// TwinCAT 3 PLC project PLC_v01
// ProgramVersion: 3.1.4022.1
// libraries:
//   Tc2_MC2, * (Beckhoff Automation GmbH)
//   Tc2_MC2_Drive, * (Beckhoff Automation GmbH)
//   Tc2_NCI, * (Beckhoff Automation GmbH)
//   Tc2_NcKinematicTransformation, * (Beckhoff Automation GmbH)
//   Tc2_Standard, * (Beckhoff Automation GmbH)
//   Tc2_System, * (Beckhoff Automation GmbH)
//   Tc2_Utilities, * (Beckhoff Automation GmbH)
//   Tc3_Module, * (Beckhoff Automation GmbH)
//   Tc3_PLCopen_OpcUa, * (Beckhoff Automation GmbH)
//   VisuDialogs, * (System)
// project tree:
//   DUTs/ E_NciChannelState.TcDUT (not stored), ST_AxisInterface.TcDUT (not stored), ST_AxisInterfaceIn.TcDUT (not stored), ST_AxisInterfaceOut.TcDUT (not stored), ST_FileDialogParams.TcDUT (not stored), ST_OpcUAVariablesR.TcDUT (not stored), ST_OpcUAVariablesW.TcDUT
//   GVLs/ GVL_Axis.TcGVL, GVL_FileOpen.TcGVL, GVL_Kin.TcGVL (not stored), GVL_Nci.TcGVL (not stored), GVL_Process.TcGVL
//   / PlcTask.TcTTO (not stored), Visualization Manager.TcVMO (not stored)
//   POUs/ FB_AxisControl.TcPOU, MAIN.TcPOU, PRG_MFuncControl.TcPOU, PRG_NcControl.TcPOU (not stored), PRG_Process.TcPOU
//   POUs/KIN/ PRG_Kinematic.TcPOU (not stored)
//   POUs/NCI/ FB_NciChannel.TcPOU, FB_NciFastMFunctions.TcPOU (not stored), FB_NciMFunctions.TcPOU, FB_NciReadLine.TcPOU, FB_NciWriteToolParams.TcPOU
//   POUs/OPC-UA/ FB_OpcUAWrite.TcPOU, PRG_OpcUA.TcPOU
//   POUs/UTIL/ FB_Flash.TcPOU, FB_ScreenOnOff_Win7.TcPOU (not stored)
//   VISUs/AxisList/ VisuAxisM1.TcVIS (not stored), VisuAxisM2.TcVIS (not stored), VisuAxisM3.TcVIS (not stored), VisuAxisX.TcVIS, VisuAxisX_1.TcVIS (not stored), VisuAxisY.TcVIS (not stored), VisuAxisY_1.TcVIS (not stored), VisuAxisZ.TcVIS, VisuAxisZ_1.TcVIS
//   VISUs/Frame/ Visualization_FileList.TcVIS (not stored), VisuAxisControl.TcVIS (not stored), VisuAxisControl_1.TcVIS (not stored), VisuAxisInfo.TcVIS
//   VISUs/ GlobalTextList.TcGTLO, ImagePool.TcIPO (not stored), Visualization.TcVIS, Visualization_AxesInfo.TcVIS (not stored), Visualization_AxesInfo_Manual.TcVIS (not stored)
// real-time tasks:
//   TASK PlcTask: cycle T#10ms, priority 20, ADS port 350
// motion (NC):
//   TASK NC-Task 1 SAF: cycle T#2ms, priority 4, ADS port 501
//   TASK NC-Task 1 SVB: cycle T#10ms, priority 8, ADS port 511
//   AXIS M1 (id 1)
//     Dynamic: Acceleration=120.483870963794, Deceleration=120.483870963794, Jerk=361.451612891381, DelayTime=0.008
//     Velo: RefSearch=0.803225806425292, RefSync=0.803225806425292, SlowManual=10, FastManual=25, Fast=80.3225806425291, Maximum=80.3225806425291
//     OtherSettings: AllowMotionCmdToSlave=true
//     encoder EncType=1
//       EncPara: ScaleFactorNumerator=11.6129032254259, ScaleFactorDenominator=1048576, Offset=-0.7867, Inverse=true
//     drive DrvType=5
//       DrvPara: Inverse=true
//         Analog: VeloReferenz=88.3548387067821, TorqueScale=10, ScaleFactorActTorque=0.1
//         TimeComp: TaskDelayCycles=1
//     controller CtrType=1
//       CtrPara: PriorControlFactor=1
//         PID: PosKp=10
//         Observer: BandWidth=20
//   AXIS M2 (id 2)
//     Dynamic: Acceleration=120.483870963794, Deceleration=120.483870963794, Jerk=361.451612891381, DelayTime=0.008
//     Velo: RefSearch=0.803225806425292, RefSync=0.803225806425292, SlowManual=10, FastManual=25, Fast=80.3225806425291, Maximum=80.3225806425291
//     OtherSettings: AllowMotionCmdToSlave=true
//     encoder EncType=1
//       EncPara: ScaleFactorNumerator=11.6129032254259, ScaleFactorDenominator=1048576, Offset=-4.6881, Inverse=true
//     drive DrvType=5
//       DrvPara: Inverse=true
//         Analog: VeloReferenz=88.3548387067821, TorqueScale=10, ScaleFactorActTorque=0.1
//         TimeComp: TaskDelayCycles=1
//     controller CtrType=1
//       CtrPara: PriorControlFactor=1
//         PID: PosKp=10
//         Observer: BandWidth=20
//   AXIS M3 (id 3)
//     Dynamic: Acceleration=120.483870963794, Deceleration=120.483870963794, Jerk=361.451612891381, DelayTime=0.008
//     Velo: RefSearch=0.803225806425292, RefSync=0.803225806425292, SlowManual=10, FastManual=25, Fast=80.3225806425291, Maximum=80.3225806425291
//     OtherSettings: AllowMotionCmdToSlave=true
//     encoder EncType=1
//       EncPara: ScaleFactorNumerator=11.6129032254259, ScaleFactorDenominator=1048576, Offset=4810.3626, Inverse=true
//     drive DrvType=5
//       DrvPara: Inverse=true
//         Analog: VeloReferenz=88.3548387067821, TorqueScale=10, ScaleFactorActTorque=0.1
//         TimeComp: TaskDelayCycles=1
//     controller CtrType=1
//       CtrPara: PriorControlFactor=1
//         PID: PosKp=10
//         Observer: BandWidth=20
//   AXIS X (id 4)
//     OtherSettings: AllowMotionCmdToSlave=true
//     encoder EncType=1
//     drive DrvType=5
//       Analog: ScaleFactorActTorque=0.1
//       TimeComp: TaskDelayCycles=1
//     controller CtrType=1
//       CtrPara: PriorControlFactor=1
//         Observer: BandWidth=20
//   AXIS Y (id 5)
//     OtherSettings: AllowMotionCmdToSlave=true
//     encoder EncType=1
//     drive DrvType=5
//       Analog: ScaleFactorActTorque=0.1
//       TimeComp: TaskDelayCycles=1
//     controller CtrType=1
//       CtrPara: PriorControlFactor=1
//         Observer: BandWidth=20
//   AXIS Z (id 6)
//     OtherSettings: AllowMotionCmdToSlave=true
//     encoder EncType=1
//     drive DrvType=5
//       Analog: ScaleFactorActTorque=0.1
//       TimeComp: TaskDelayCycles=1
//     controller CtrType=1
//       CtrPara: PriorControlFactor=1
//         Observer: BandWidth=20
// I/O:
//   DEVICE Device 1 (EtherCAT) (disabled), AmsNetId 10.70.16.23.2.1
//     Term 1 (EK1200) [EK1200-5000 EtherCAT Power supply (2A E-Bus)]
//       Term 2 (EL1008) [EL1008 8Ch. Dig. Input 24V, 3ms]
//       Term 3 (EL2008) [EL2008 8Ch. Dig. Output 24V, 0.5A]
//       Term 4 (EL9576) [EL9576 Brake chopper terminal]
//       Term 5 (EL7211-0010) [EL7211-0010 1Ch. MDP742 Servo motor output stage with OCT (50V, 4.5A RMS)]
//       Term 6 (EL7211-0010) [EL7211-0010 1Ch. MDP742 Servo motor output stage with OCT (50V, 4.5A RMS)]
//       Term 7 (EL7211-0010) [EL7211-0010 1Ch. MDP742 Servo motor output stage with OCT (50V, 4.5A RMS)]
//       Term 8 (EL9011) [EL9011 End Terminal]
// variable links:
//   PLC_v01/PLC_v01 Instance <-> NC-Task 1 SAF/Axes/M1
//     PlcTask Inputs/GVL_Axis.AxisM1_B.NcToPlc <-> Outputs/ToPlc
//     PlcTask Outputs/GVL_Axis.AxisM1_B.PlcToNc <-> Inputs/FromPlc
//   PLC_v01/PLC_v01 Instance <-> NC-Task 1 SAF/Axes/M2
//     PlcTask Inputs/GVL_Axis.AxisM2_C.NcToPlc <-> Outputs/ToPlc
//     PlcTask Outputs/GVL_Axis.AxisM2_C.PlcToNc <-> Inputs/FromPlc
//   PLC_v01/PLC_v01 Instance <-> NC-Task 1 SAF/Axes/M3
//     PlcTask Inputs/GVL_Axis.AxisM3_A.NcToPlc <-> Outputs/ToPlc
//     PlcTask Outputs/GVL_Axis.AxisM3_A.PlcToNc <-> Inputs/FromPlc
//   PLC_v01/PLC_v01 Instance <-> NC-Task 1 SAF/Axes/X
//     PlcTask Inputs/GVL_Axis.AxisX.NcToPlc <-> Outputs/ToPlc
//     PlcTask Outputs/GVL_Axis.AxisX.PlcToNc <-> Inputs/FromPlc
//   PLC_v01/PLC_v01 Instance <-> NC-Task 1 SAF/Axes/Y
//     PlcTask Inputs/GVL_Axis.AxisY.NcToPlc <-> Outputs/ToPlc
//     PlcTask Outputs/GVL_Axis.AxisY.PlcToNc <-> Inputs/FromPlc
//   PLC_v01/PLC_v01 Instance <-> NC-Task 1 SAF/Axes/Z
//     PlcTask Inputs/GVL_Axis.AxisZ.NcToPlc <-> Outputs/ToPlc
//     PlcTask Outputs/GVL_Axis.AxisZ.PlcToNc <-> Inputs/FromPlc
//   PLC_v01/PLC_v01 Instance <-> NC-Task 1 SAF/KIN
//     PlcTask Inputs/GVL_Kin.stKinToPLC <-> Outputs/ToPlc
//     PlcTask Outputs/GVL_Kin.stKinFromPLC <-> Inputs/FromPlc
//   PLC_v01/PLC_v01 Instance <-> NC-Task 1 SAF/NCI
//     PlcTask Inputs/GVL_Nci.stNciToPLC <-> Outputs/ToPlc
//     PlcTask Outputs/GVL_Nci.stPlcToNci <-> Inputs/FromPlc

// ---- DUTs/ST_OpcUAVariablesW.TcDUT
TYPE ST_OpcUAVariablesW :
STRUCT
	fActPosX		: LREAL;
	fActPosY		: LREAL;
	fActPosZ		: LREAL;
	fActPosM1		: LREAL;
	fActPosM2		: LREAL;
	fActPosM3		: LREAL;
	
	fActVeloX		: LREAL;
	fActVeloY		: LREAL;
	fActVeloZ		: LREAL;
	fActVeloM1		: LREAL;
	fActVeloM2		: LREAL;
	fActVeloM3		: LREAL;
	
	fLagDistanceX	: LREAL;
	fLagDistanceY	: LREAL;
	fLagDistanceZ	: LREAL;
	fLagDistanceM1	: LREAL;
	fLagDistanceM2	: LREAL;
	fLagDistanceM3	: LREAL;
	
	sNciActLine		: STRING;
	sNciLines		: STRING;
	sFileNameVisu	: STRING;
	
	bEnabledX		: BOOL;
	bEnabledY		: BOOL;
	bEnabledZ		: BOOL;
	bEnabledM1		: BOOL;
	bEnabledM2		: BOOL;
	bEnabledM3		: BOOL;
		
	bNciRunning		: BOOL;
	bNciStopped		: BOOL;
	bNciFinished	: BOOL;

	bErrorX			: BOOL;
	bErrorY			: BOOL;
	bErrorZ			: BOOL;
	bErrorM1		: BOOL;
	bErrorM2		: BOOL;
	bErrorM3		: BOOL;
	
END_STRUCT
END_TYPE

// ---- GVLs/GVL_Axis.TcGVL
VAR_GLOBAL
// Kullanilacak olan gercek eksenler
	AxisM1_B			: AXIS_REF;			
	AxisM2_C			: AXIS_REF;
	AxisM3_A			: AXIS_REF;	
	
// Kinematik grupta olusacak eksenler
	AxisX				: AXIS_REF;
	AxisY				: AXIS_REF;
	AxisZ				: AXIS_REF;
	
// Gercek eksenler icin interface yapilari
	stAxisM1_B			: ST_AxisInterface;
	stAxisM2_C			: ST_AxisInterface;
	stAxisM3_A			: ST_AxisInterface;
	
// Kinematik eksenlerin interface yapilari
	stAxisX				: ST_AxisInterface;
	stAxisY				: ST_AxisInterface;
	stAxisZ				: ST_AxisInterface;
	
	sAxisM1_BName		: STRING	:= 'Axis M1';
	sAxisM2_CName		: STRING	:= 'Axis M2';
	sAxisM3_AName		: STRING	:= 'Axis M3';
	
	
	sAxisXName			: STRING	:= 'Axis X';
	sAxisYName			: STRING	:= 'Axis Y';
	sAxisZName			: STRING	:= 'Axis Z';
	
	AxisM1PosValue		: LREAL;
	AxisM2PosValue		: LREAL;
	AxisM3PosValue		: LREAL;
	
	AxisM1VeloValue		: LREAL;
	AxisM2VeloValue		: LREAL;
	AxisM3VeloValue		: LREAL;
	
END_VAR

// ---- GVLs/GVL_FileOpen.TcGVL
{attribute 'qualified_only'}
VAR_GLOBAL
	fbFileListProvider	: Visu_FbFileListProvider;
	stFileDialogParams 	: ST_FileDialogParams;
	bFileDialogOpen 	: BOOL := FALSE;
 
END_VAR

// ---- GVLs/GVL_Process.TcGVL
{attribute 'qualified_only'}
VAR_GLOBAL
	bAllAxesEnablePLC	: BOOL;
	bAllAxesEnable		: BOOL;
	bAllAxesEnabled		: BOOL;
	bAllAxesReset		: BOOL;
	bNciStartPLC		: BOOL;
	
	bEmergencyOnPanel 	AT%I*	: BOOL;
	fTrigbEmergency				: F_TRIG;
	rTrigbEmergency				: R_TRIG;
	bGreenBtnOnPanel	AT%I*	: BOOL;
	nStateEmergency				: INT;
	
	bManualSelectX		: BOOL;
	bManualSelectY		: BOOL;
	bManualSelectZ		: BOOL;
	nSizeSelectX		: INT := 27;
	nSizeSelectY		: INT := 27;
	nSizeSelectZ		: INT := 27;
	
	nAutoManMode		: BOOL;
	
	bMessageBubbleAuto	: BOOL;
	bMessageBubbleMan	: BOOL;
	
	stOpcUaVariablesW	: ST_OpcUAVariablesW;
	stOpcUaVariablesR	: ST_OpcUAVariablesR;
END_VAR

// ---- POUs/FB_AxisControl.TcPOU
FUNCTION_BLOCK FB_AxisControl
VAR_IN_OUT
	stAxisInterface		: ST_AxisInterface;
	stAxisRef			: AXIS_REF;
END_VAR
VAR
	fbPower				: MC_Power;
	fbReset				: MC_Reset;
	fbDriveReset		: FB_SoeReset;
	fbHome				: MC_Home;
	fbReadStatus		: MC_ReadStatus;
	fbMoveAbsoluteP1	: MC_MoveAbsolute;
	fbMoveAbsoluteP2	: MC_MoveAbsolute;
	fbStop				: MC_Stop;
	fbJog				: MC_Jog;
	fbResetTrig			: R_TRIG;
	fbDriveResetTrig	: R_TRIG;
	fbHomeFallTrig		: F_TRIG;
	fbMoveFallTrig		: F_TRIG;
	nState				: INT;
	bAxisOk				: BOOL;
	fOldSetPos			: LREAL;
END_VAR


(* Enable Axis		*)
fbPower(
	Axis			:= stAxisRef, 
	Enable			:= stAxisInterface.In.xEnable, 
	Enable_Positive	:= stAxisInterface.In.xEnable, 
	Enable_Negative	:= stAxisInterface.In.xEnable, 
	Override		:= stAxisInterface.In.fOverride,
	Status			=> stAxisInterface.Out.xEnabled );
(***********************************************************)

(* Reset Axis 		*)
fbResetTrig(CLK:= stAxisInterface.In.xReset);
fbReset(
	Axis			:= stAxisRef, 
	Execute			:= fbResetTrig.Q );
(***********************************************************)
	
(* Reset Drive		*)
fbDriveResetTrig(CLK:= stAxisInterface.In.xDriveReset);
fbDriveReset(
	NetId			:= '', 
	Execute			:= fbDriveResetTrig.Q, 
	Timeout			:= T#5S, 
	Axis			:= stAxisRef );
(***********************************************************)
	
(* Read Status		*)
stAxisRef.ReadStatus();
fbReadStatus(
	Axis			:= stAxisRef, 
	Enable			:= TRUE, 
	Error			=> stAxisInterface.Out.xAxisError, 
	ErrorID			=> stAxisInterface.Out.nAxisErrId );
	
bAxisOk				:= (NOT stAxisInterface.Out.xAxisError) AND stAxisInterface.Out.xEnabled;
(***********************************************************)
	
(* Home				*)
fbHome(
	Axis			:= stAxisRef, 
	Execute			:= stAxisInterface.In.xHome AND bAxisOk, 
	Position		:= stAxisInterface.In.fHomePos, 
	bCalibrationCam	:= stAxisInterface.In.xHomeSensor, 
	Done			=> stAxisInterface.Out.xHomed);
(***********************************************************)
	
(* Jog				*)
fbJog(
	Axis			:= stAxisRef, 
	JogForward		:= stAxisInterface.In.xJogFw AND bAxisOk, 
	JogBackwards	:= stAxisInterface.In.xJogBw AND bAxisOk, 
	Mode			:= MC_JOGMODE_CONTINOUS, 
	Velocity		:= stAxisInterface.In.fJogVelo );
(***********************************************************)
	
(* Move	Absolute	*)
fbMoveAbsoluteP1(
	Axis			:= stAxisRef, 
	Execute			:= fbMoveAbsoluteP1.Execute AND bAxisOk, 
	Position		:= fbMoveAbsoluteP1.Position, 
	Velocity		:= fbMoveAbsoluteP1.Velocity, 
	Acceleration	:= fbMoveAbsoluteP1.Acceleration, 
	Deceleration	:= fbMoveAbsoluteP1.Deceleration, 
	Jerk			:= fbMoveAbsoluteP1.Jerk,
	BufferMode   	:= MC_Aborting );
	
fbMoveAbsoluteP2(
	Axis			:= stAxisRef, 
	Execute			:= fbMoveAbsoluteP2.Execute AND bAxisOk, 
	Position		:= fbMoveAbsoluteP2.Position, 
	Velocity		:= fbMoveAbsoluteP2.Velocity, 
	Acceleration	:= fbMoveAbsoluteP2.Acceleration, 
	Deceleration	:= fbMoveAbsoluteP2.Deceleration, 
	Jerk			:= fbMoveAbsoluteP2.Jerk,
	BufferMode   	:= MC_Aborting );

CASE nState OF
	
0:
	stAxisInterface.Out.xMoveDone	:= FALSE;
	fbMoveAbsoluteP1.Execute		:= FALSE;
	fbMoveAbsoluteP2.Execute		:= FALSE;
	
	IF bAxisOK AND stAxisInterface.In.xMove THEN
		fbMoveAbsoluteP1.Position		:= stAxisInterface.In.fSetPos;
		fbMoveAbsoluteP1.Velocity		:= stAxisInterface.In.fSetVelo;
		fbMoveAbsoluteP1.Acceleration	:= stAxisInterface.In.fSetAcc;
		fbMoveAbsoluteP1.Deceleration	:= stAxisInterface.In.fSetDec;
		fOldSetPos						:= stAxisInterface.In.fSetPos;
		fbMoveAbsoluteP1.Execute		:= TRUE;
		nState	:= 10;
	END_IF
	
10:
	IF fbMoveAbsoluteP1.Done THEN
		stAxisInterface.Out.xMoveDone	:= TRUE;
		nState	:= 30;
	ELSE
		IF fOldSetPos <> stAxisInterface.In.fSetPos THEN
			stAxisInterface.Out.xMoveDone	:= FALSE;
			fbMoveAbsoluteP1.Execute		:= FALSE;
			fbMoveAbsoluteP2.Position		:= stAxisInterface.In.fSetPos;
			fbMoveAbsoluteP2.Velocity		:= stAxisInterface.In.fSetVelo;
			fbMoveAbsoluteP2.Acceleration	:= stAxisInterface.In.fSetAcc;
			fbMoveAbsoluteP2.Deceleration	:= stAxisInterface.In.fSetDec;
			fOldSetPos						:= stAxisInterface.In.fSetPos;
			fbMoveAbsoluteP2.Execute		:= TRUE;
			nState	:= 20;
		END_IF
	END_IF
	
20:
	IF fbMoveAbsoluteP2.Done THEN
		stAxisInterface.Out.xMoveDone	:= TRUE;
		nState	:= 30;
	ELSE
		IF fOldSetPos <> stAxisInterface.In.fSetPos THEN
			stAxisInterface.Out.xMoveDone	:= FALSE;
			fbMoveAbsoluteP2.Execute		:= FALSE;
			fbMoveAbsoluteP1.Position		:= stAxisInterface.In.fSetPos;
			fbMoveAbsoluteP1.Velocity		:= stAxisInterface.In.fSetVelo;
			fbMoveAbsoluteP1.Acceleration	:= stAxisInterface.In.fSetAcc;
			fbMoveAbsoluteP1.Deceleration	:= stAxisInterface.In.fSetDec;
			fOldSetPos						:= stAxisInterface.In.fSetPos;
			fbMoveAbsoluteP1.Execute		:= TRUE;
			nState	:= 10;
		END_IF
	END_IF
	
30:
	fbMoveAbsoluteP1.Execute		:= FALSE;
	fbMoveAbsoluteP2.Execute		:= FALSE;
	
	IF NOT stAxisInterface.In.xMove THEN
		stAxisInterface.Out.xMoveDone	:= FALSE;
		nState	:= 0;
	ELSE
		IF fOldSetPos <> stAxisInterface.In.fSetPos THEN
			stAxisInterface.Out.xMoveDone	:= FALSE;
			nState	:= 10;
		END_IF
	END_IF

END_CASE

(***********************************************************)

(* Stop				*)
fbHomeFallTrig(CLK:= stAxisInterface.In.xHome);
fbMoveFallTrig(CLK:= stAxisInterface.In.xMove);
fbStop(
	Axis			:= stAxisRef, 
	Execute			:= fbMoveFallTrig.Q OR fbHomeFallTrig.Q);
	
(* Function Error	*)
IF fbPower.Error THEN
	stAxisInterface.Out.xFunctionError	:= fbPower.Error;
	stAxisInterface.Out.nFunctionErrId	:= fbPower.ErrorID;
ELSIF fbReset.Error THEN
	stAxisInterface.Out.xFunctionError	:= fbReset.Error;
	stAxisInterface.Out.nFunctionErrId	:= fbReset.ErrorID;
ELSIF fbDriveReset.Error THEN
	stAxisInterface.Out.xFunctionError	:= fbDriveReset.Error;
	stAxisInterface.Out.nFunctionErrId	:= fbDriveReset.AdsErrId;
ELSIF fbHome.Error THEN
	stAxisInterface.Out.xFunctionError	:= fbHome.Error;
	stAxisInterface.Out.nFunctionErrId	:= fbHome.ErrorID;
ELSIF fbJog.Error THEN
	stAxisInterface.Out.xFunctionError	:= fbJog.Error;
	stAxisInterface.Out.nFunctionErrId	:= fbJog.ErrorID;
ELSIF fbMoveAbsoluteP1.Error THEN
	stAxisInterface.Out.xFunctionError	:= fbMoveAbsoluteP1.Error;
	stAxisInterface.Out.nFunctionErrId	:= fbMoveAbsoluteP1.ErrorID;
ELSIF fbMoveAbsoluteP2.Error THEN
	stAxisInterface.Out.xFunctionError	:= fbMoveAbsoluteP2.Error;
	stAxisInterface.Out.nFunctionErrId	:= fbMoveAbsoluteP2.ErrorID;
ELSIF fbStop.Error THEN
	stAxisInterface.Out.xFunctionError	:= fbStop.Error;
	stAxisInterface.Out.nFunctionErrId	:= fbStop.ErrorID;
ELSE
	stAxisInterface.Out.xFunctionError	:= FALSE;
	stAxisInterface.Out.nFunctionErrId	:= 0;
END_IF

END_FUNCTION_BLOCK

// ---- POUs/MAIN.TcPOU
PROGRAM MAIN
VAR
	sFilePathName	: STRING := 'C:\TwinCAT\CNC\TestNci1.txt';
	sErrorMessage	: STRING := '';
	bOpen			: BOOL;
	bClose 			: BOOL;
	bSave 			: BOOL;
	bNew			: BOOL;
	nErrorCode		: USINT;
	nLineNumber		: USINT;
	bEnable: BOOL;
END_VAR

(*V03 	- 28.09.2017 13:40*)
(*V03.1 - 10.02.2017 *)

sErrorMessage	:= VisuFctTextEditorGetErrorText(usiErrCode := nErrorCode);

PRG_NcControl();
//PRG_MFuncControl();
PRG_Kinematic();

//PRG_Process();

//PRG_OpcUA();


IF bEnable THEN
	stAxisM1_B.In.xEnable	:= TRUE;
	stAxisM2_C.In.xEnable	:= TRUE;
	stAxisM3_A.In.xEnable	:= TRUE;
	stAxisX.In.xEnable	:= TRUE;
	stAxisY.In.xEnable	:= TRUE;
	stAxisZ.In.xEnable	:= TRUE;
	
	stAxisM1_B.In.fOverride	:= 100;
	stAxisM2_C.In.fOverride	:= 100;
	stAxisM3_A.In.fOverride	:= 100;
	stAxisX.In.fOverride	:= 100;
	stAxisY.In.fOverride	:= 100;
	stAxisZ.In.fOverride	:= 100;
ELSE
	stAxisM1_B.In.xEnable	:= FALSE;
	stAxisM2_C.In.xEnable	:= FALSE;
	stAxisM3_A.In.xEnable	:= FALSE;
	stAxisX.In.xEnable	:= FALSE;
	stAxisY.In.xEnable	:= FALSE;
	stAxisZ.In.xEnable	:= FALSE;
END_IF

stAxisX.In.fSetPos;
stAxisY.In.fSetPos;
stAxisZ.In.fSetPos;

stAxisX.In.fSetVelo;
stAxisY.In.fSetVelo;
stAxisZ.In.fSetVelo;

stAxisX.In.xMove;
stAxisY.In.xMove;
stAxisZ.In.xMove;


AxisM1PosValue	:= AxisM1_B.NcToPlc.ActPos;
AxisM2PosValue	:= AxisM2_C.NcToPlc.ActPos;
AxisM3PosValue	:= AxisM3_A.NcToPlc.ActPos;

AxisM1VeloValue	:= AxisM1_B.NcToPlc.ActVelo;
AxisM2VeloValue	:= AxisM2_C.NcToPlc.ActVelo;
AxisM3VeloValue	:= AxisM3_A.NcToPlc.ActVelo;

END_PROGRAM

// ---- POUs/NCI/FB_NciChannel.TcPOU
FUNCTION_BLOCK FB_NciChannel
VAR_INPUT
	bEnable				: BOOL;
	bStart				: BOOL;
	bSingleMode			: BOOL;
	bSingleModeStart	: BOOL;
	fOverride			: LREAL;
	nXAxisId			: UDINT;
	nYAxisId			: UDINT;
	nZAxisId			: UDINT;
	sProgramPath		: STRING(255);
	sSubroutinePath		: STRING(255);
END_VAR
VAR_IN_OUT
	sNciToPLC			: NCTOPLC_NCICHANNEL_REF;
	sPlcToNci			: PLCTONC_NCICHANNEL_REF;
END_VAR
VAR_OUTPUT
	eNciChannelState	: E_NciChannelState;
	bBuildGroupDone		: BOOL;
	bSingleModeActive	: BOOL;
	bProgramRunning		: BOOL;
	bProgramStopped		: BOOL;
	bProgramFinished	: BOOL;
	bError				: BOOL;
	nErrorId			: UDINT;
END_VAR
VAR
	fbNciReset			: ItpResetEx2;
	fbBuildGroup		: CfgBuildExt3DGroup;
	fbSetSubroutinePath	: ItpSetSubroutinePathEx;
	fbLoadProgram		: ItpLoadProgEx;
	fbStartStop			: ItpStartStopEx;
	fbEStop				: ItpEStopEx;
	fbStepOnAfterEStop	: ItpStepOnAfterEStopEx;
	fbConfirmMFunc		: ItpConfirmHsk;
	fbClearGroup		: CfgReconfigGroup;
	fbReadRParams		: ItpReadRParamsEx;
	fbWriteRParams		: ItpWriteRParamsEx;
	fbReadToolDesc		: ItpReadToolDescEx;
	fbWriteToolDesc		: FB_NciWriteToolParams;
	fbSingleBlock		: ItpSingleBlock;
	nSingleMode			: E_ItpSingleBlockMode;
	rTrigNext			: R_TRIG;
	nItpState			: UDINT;
	nState				: INT;
	nLastState			: INT;
	bConfirmMFunc		: BOOL;
END_VAR

(* Set NCI Channel Override	*)
ItpSetOverridePercent(fOverridePercent:= fOverride, sPlcToNci:= sPlcToNci );

(* Get Actual Channel State	*)
nItpState			:= ItpGetStateInterpreter(sNciToPlc:= sNciToPlc);
eNciChannelState	:= UDINT_TO_INT(nItpState);

(* Single Mode Selection	*)
IF bSingleMode THEN
	nSingleMode	:= ItpSingleBlockIntp;
ELSE
	nSingleMode	:= ItpSingleBlockOff;
END_IF


CASE nState OF
	
0:
	bBuildGroupDone		:= FALSE;
	bSingleModeActive	:= FALSE;
	bProgramRunning		:= FALSE;
	bProgramStopped		:= FALSE;
	bProgramFinished	:= FALSE;
	bError				:= FALSE;
	nErrorId			:= 0;
	
	IF bEnable THEN
		nState		:= 10;
		nLastState	:= nState;
	END_IF
	
10:
	(* Reset NCI First	*)
	fbNciReset(
		bExecute	:= TRUE, 
		tTimeOut	:= T#500MS, 
		sNciToPlc	:= sNciToPLC );
		
	IF NOT fbNciReset.bBusy AND NOT fbNciReset.bErr THEN
		fbNciReset(bExecute := FALSE, sNciToPlc := sNciToPLC);
		nState		:= 20;
		nLastState	:= nState;
	ELSIF fbNciReset.bErr THEN
		fbNciReset(bExecute := FALSE, sNciToPlc := sNciToPLC);
		bError		:= TRUE;
		nErrorId	:= fbNciReset.nErrId;
		nState		:= 9000;
	END_IF
	
20:
	(* Build NCI Group	*)
	fbBuildGroup(
		bExecute	:= TRUE, 
		nGroupId	:= ItpGetGroupId(sNciToPlc:= sNciToPlc), 
		nXAxisId	:= nXAxisId, 
		nYAxisId	:= nYAxisId, 
		nZAxisId	:= nZAxisId, 
		tTimeOut	:= T#500MS );
		
	IF NOT fbBuildGroup.bBusy AND NOT fbBuildGroup.bErr THEN
		fbBuildGroup(bExecute := FALSE);
		bBuildGroupDone	:= TRUE;
		nState		:= 30;
		nLastState	:= nState;
	ELSIF fbBuildGroup.bErr THEN
		fbBuildGroup(bExecute := FALSE);
		bError		:= TRUE;
		nErrorId	:= fbBuildGroup.nErrId;
		nState		:= 9000;
	END_IF
	
30:
	(* Set NCI Subroutine Path	*)
	fbSetSubroutinePath(
		bExecute	:= TRUE, 
		sPath		:= sSubroutinePath, 
		nLength		:= INT_TO_UDINT(LEN(sSubroutinePath)), 
		tTimeOut	:= T#500MS, 
		sNciToPlc	:= sNciToPLC);
		
	IF NOT fbSetSubroutinePath.bBusy AND NOT fbSetSubroutinePath.bErr THEN
		fbSetSubroutinePath(bExecute := FALSE, sNciToPlc := sNciToPLC);
		nState		:= 40;
		nLastState	:= nState;
	ELSIF fbSetSubroutinePath.bErr THEN
		fbSetSubroutinePath(bExecute := FALSE, sNciToPlc := sNciToPLC);
		bError		:= TRUE;
		nErrorId	:= fbSetSubroutinePath.nErrId;
		nState		:= 9000;
	END_IF
	
40:
	(* If start then jump to state 100*)
	IF bEnable THEN
		IF bStart THEN
			nState		:= 100;
			nLastState	:= nState;
		END_IF
	ELSE
		nState		:= 300;
		nLastState	:= nState;
	END_IF
	
100:
	(* Write R Params before load the program	*)
	fbWriteRParams(
		bExecute	:= TRUE, 
		pAddr		:= ADR(fNciRParamsWrite), 
		nIndex		:= cnStartIndexWriteRParam, 
		nCount		:= (cnEndIndexWriteRParam - cnStartIndexWriteRParam) + 1, 
		tTimeOut	:= T#200MS, 
		sNciToPlc	:= sNciToPLC );	
		
	IF NOT fbWriteRParams.bBusy AND NOT fbWriteRParams.bErr THEN
		fbWriteRParams( bExecute := FALSE, sNciToPlc := sNciToPLC);
		nState		:= 110;
		nLastState	:= nState;
	ELSIF fbWriteRParams.bErr THEN
		fbWriteRParams( bExecute := FALSE, sNciToPlc := sNciToPLC);
		bError		:= TRUE;
		nErrorId	:= fbWriteRParams.nErrId;
		nState		:= 9000;
	END_IF
	
110:
	(* Write Tool Params before load the program	*)
	fbWriteToolDesc(
		bExecute	:= TRUE, 
		sNciToPLC	:= sNciToPLC );
		
	IF fbWriteToolDesc.bDone THEN
		fbWriteToolDesc(bExecute := FALSE, sNciToPlc := sNciToPLC);
		nState		:= 120;
		nLastState	:= nState;
	ELSIF fbWriteToolDesc.bError THEN
		fbWriteToolDesc(bExecute := FALSE, sNciToPlc := sNciToPLC);
		bError		:= TRUE;
		nErrorId	:= fbWriteToolDesc.nErrorId;
		nState		:= 9000;
	END_IF
	
120:
	(* Load Program	*)
	fbLoadProgram(
		sNciToPlc	:= sNciToPlc, 
		bExecute	:= TRUE, 
		sPrg		:= sProgramPath, 
		nLength		:= INT_TO_UDINT(LEN(sProgramPath)), 
		tTimeOut	:= T#500MS);
		
	IF NOT fbLoadProgram.bBusy AND NOT fbLoadProgram.bErr THEN
		fbLoadProgram(bExecute := FALSE, sNciToPlc := sNciToPLC);
		nState		:= 130;
		nLastState	:= nState;
	ELSIF fbLoadProgram.bErr THEN
		fbLoadProgram(bExecute := FALSE, sNciToPlc := sNciToPLC);
		bError		:= TRUE;
		nErrorId	:= fbLoadProgram.nErrId;
		nState		:= 9000;
	END_IF
	
130:
	(* Be sure fbStartStop FALSE	*)
	fbStartStop(
		bStart		:= FALSE, 
		bStop		:= FALSE, 
		tTimeOut	:= T#500MS, 
		sNciToPlc	:= sNciToPlc);

	IF nItpState = NCI_INTERPRETER_READY THEN
		nState		:= 140;
		nLastState	:= nState;
	ELSIF nItpState = NCI_INTERPRETER_ABORTED THEN
		bError		:= TRUE;
		nErrorId	:= 4711;
		nState		:= 9000;
	END_IF
	
140:
	(* Set SingleBlock Mode		*)
	fbSingleBlock(
		bExecuteModeChange	:= TRUE, 
		nMode				:= nSingleMode, 
		bTriggerNext		:= FALSE, 
		tTimeOut			:= T#100MS, 
		sNciToPlc			:= sNciToPlc );
	
	rTrigNext(CLK:= FALSE);
	
	IF NOT fbSingleBlock.bBusy AND NOT fbSingleBlock.bErr THEN
		fbSingleBlock(bExecuteModeChange := FALSE, sNciToPlc := sNciToPlc);
		IF NOT bSingleMode THEN
			nState		:= 150;
			nLastState	:= nState;
		ELSE
			nState		:= 170;
			nLastState	:= nState;
		END_IF
	ELSIF fbSingleBlock.bErr THEN
		fbSingleBlock(bExecuteModeChange := FALSE, sNciToPlc := sNciToPlc);
		bError		:= TRUE;
		nErrorId	:= fbSingleBlock.nErrId;
		nState		:= 9000;
	END_IF
	
150:
	(* If not single block mode run	*)
	fbStartStop(
		bStart		:= TRUE, 
		bStop		:= FALSE, 
		tTimeOut	:= T#500MS, 
		sNciToPlc	:= sNciToPlc);
		
	IF NOT fbStartStop.bBusy AND NOT fbStartStop.bErr THEN
		fbStartStop(bStart := FALSE, bStop := FALSE, sNciToPlc := sNciToPLC);
		nState		:= 160;
		nLastState	:= nState;
	ELSIF fbStartStop.bErr THEN
		fbStartStop(bStart := FALSE, bStop := FALSE, sNciToPlc := sNciToPLC);
		bError		:= TRUE;
		nErrorId	:= fbLoadProgram.nErrId;
		nState		:= 9000;
	END_IF
	
160:
	(* Check if the channel running	*)
	IF bEnable THEN
		(* Check if the part program is really started!*)
		(* If the part program finished without an error, 
			then it switch back to ready state *)
		IF nItpState <> NCI_INTERPRETER_READY THEN
			bProgramRunning	:= TRUE;
			nState		:= 200;
			nLastState	:= nState;
		END_IF
	ELSE
		nState		:= 300;
		nLastState	:= nState;
	END_IF
	
170:
	(* Activate single block mode	*)
	rTrigNext(CLK:= TRUE);

	fbSingleBlock(
		bExecuteModeChange	:= FALSE, 
		nMode				:= nSingleMode, 
		bTriggerNext		:= rTrigNext.Q, 
		tTimeOut			:= T#100MS, 
		sNciToPlc			:= sNciToPlc );
		
	IF nItpState = NCI_INTERPRETER_SINGLESTOP THEN
		rTrigNext(CLK:= FALSE);
		bSingleModeActive	:= TRUE;
		nState		:= 180;
		nLastState	:= nState;
	END_IF
	
180:
	(* With next click run the program line by line	*)
	rTrigNext(CLK:= bSingleModeStart AND bSingleMode);

	fbSingleBlock(
		bExecuteModeChange	:= FALSE, 
		nMode				:= nSingleMode, 
		bTriggerNext		:= rTrigNext.Q, 
		tTimeOut			:= T#100MS, 
		sNciToPlc			:= sNciToPlc );
	
	IF nItpState = NCI_INTERPRETER_READY THEN
		bProgramRunning		:= FALSE;
		bProgramStopped		:= FALSE;
		bProgramFinished	:= TRUE;
		nState		:= 190;
		nLastState	:= nState;
	END_IF
		
	IF NOT bSingleMode THEN
		nState		:= 190;
		nLastState	:= nState;
	END_IF
	
190:
	(* Turn off the single block mode	*)
	fbSingleBlock(
		bExecuteModeChange	:= TRUE, 
		nMode				:= ItpSingleBlockOff, 
		bTriggerNext		:= FALSE, 
		tTimeOut			:= T#100MS, 
		sNciToPlc			:= sNciToPlc );
		
	IF NOT fbSingleBlock.bBusy AND NOT fbSingleBlock.bErr THEN
		fbSingleBlock(bExecuteModeChange := FALSE, sNciToPlc := sNciToPlc);
		bSingleModeActive	:= FALSE;
		(* If program finished*)
		IF bProgramFinished THEN
			nState		:= 195;
			nLastState	:= nState;
		ELSE
		(* If program not finished*)
			bProgramRunning	:= TRUE;
			nState		:= 200;
			nLastState	:= nState;
		END_IF
	ELSIF fbSingleBlock.bErr THEN
		fbSingleBlock(bExecuteModeChange := FALSE, sNciToPlc := sNciToPlc);
		bError		:= TRUE;
		nErrorId	:= fbSingleBlock.nErrId;
		nState		:= 9000;
	END_IF
	
195:
	(* Check for start if TRUE	*)
	IF NOT bStart THEN
		bProgramFinished	:= FALSE;
		nState		:= 310;
		nLastState	:= nState;
	END_IF
	
200:
	(* Check if the program finished or stopped *)
	IF bEnable THEN
		IF (NOT bStart) THEN
			IF (NOT bProgramFinished) THEN
				bProgramStopped	:= TRUE;
				nState		:= 210;
				nLastState	:= nState;
			ELSE
				nState		:= 300;
				nLastState	:= nState;
			END_IF
		ELSE
			IF nItpState = NCI_INTERPRETER_READY OR nItpState = NCI_INTERPRETER_IDLE THEN
				bProgramRunning		:= FALSE;
				bProgramStopped		:= FALSE;
				bProgramFinished	:= TRUE;
			END_IF
		END_IF
	ELSE
		bProgramRunning	:= FALSE;
		bProgramStopped	:= FALSE;
		nState		:= 300;
		nLastState	:= nState;
	END_IF

210:
	(* Stop the channel	*)
	fbEStop(
		sNciToPlc	:= sNciToPlc, 
		bExecute	:= TRUE, 
		fDec		:= 40000, 
		fJerk		:= 400000, 
		tTimeOut	:= T#500MS);
		
	IF NOT fbEStop.bBusy AND NOT fbEStop.bErr THEN
		fbEStop(bExecute := FALSE, sNciToPlc := sNciToPLC);
		nState		:= 220;
		nLastState	:= nState;
	ELSIF fbEStop.bErr THEN
		fbEStop(bExecute := FALSE, sNciToPlc := sNciToPLC);
		bError		:= TRUE;
		nErrorId	:= fbEStop.nErrId;
		nState		:= 9000;
	END_IF

220:
	(* Decide to go on or clear the group	*)
	IF bEnable THEN
		IF bStart THEN
			nState		:= 230;
			nLastState	:= nState;
		END_IF
	ELSE
		bProgramRunning	:= FALSE;
		bProgramStopped	:= FALSE;
		nState		:= 300;
		nLastState	:= nState;
	END_IF

230:
	(* Go on *)
	fbStepOnAfterEStop(
		bExecute	:= TRUE, 
		tTimeOut	:= T#500MS, 
		sNciToPlc	:= sNciToPlc);
		
	IF NOT fbStepOnAfterEStop.bBusy AND NOT fbStepOnAfterEStop.bErr THEN
		fbStepOnAfterEStop(bExecute := FALSE, sNciToPlc := sNciToPLC);
		bProgramStopped	:= FALSE;
		nState		:= 200;
		nLastState	:= nState;
	ELSIF fbStepOnAfterEStop.bErr THEN
		fbStepOnAfterEStop(bExecute := FALSE, sNciToPlc := sNciToPLC);
		bError		:= TRUE;
		nErrorId	:= fbStepOnAfterEStop.nErrId;
		nState		:= 9000;
	END_IF
	
300:
	(* Program finished	*)
	bProgramFinished	:= FALSE;
	bProgramStopped		:= FALSE;
	bProgramRunning		:= FALSE;

	fbStartStop(
		bStart		:= FALSE, 
		bStop		:= TRUE, 
		tTimeOut	:= T#500MS, 
		sNciToPlc	:= sNciToPlc);
		
	IF NOT fbStartStop.bBusy AND NOT fbStartStop.bErr THEN
		fbStartStop(bStart := FALSE, bStop := FALSE, sNciToPlc := sNciToPLC);
		nState		:= 310;
		nLastState	:= nState;
	ELSIF fbStartStop.bErr THEN
		fbStartStop(bStart := FALSE, bStop := FALSE, sNciToPlc := sNciToPLC);
		bError		:= TRUE;
		nErrorId	:= fbLoadProgram.nErrId;
		nState		:= 9000;
	END_IF

310:
	(* InCase of any error confirm M Functions	*)
	IF (ItpGetHskMFunc(sNciToPlc:= sNciToPlc)) > 0 THEN
		bConfirmMFunc	:= TRUE;
	ELSE
		bConfirmMFunc	:= FALSE;
	END_IF
	
	fbConfirmMFunc(bExecute:= bConfirmMFunc, sNciToPlc:= sNciToPlc, sPlcToNci:= sPlcToNci);
	
	IF NOT fbConfirmMfunc.bBusy AND NOT fbConfirmMFunc.bErr THEN
		fbConfirmMFunc(bExecute:= FALSE, sNciToPlc:= sNciToPlc, sPlcToNci:= sPlcToNci);
		bConfirmMFunc	:= FALSE;
		IF bEnable THEN
			nState		:= 320;
			nLastState	:= nState;
		ELSE
			nState		:= 400;
			nLastState	:= nState;
		END_IF
	ELSIF fbConfirmMfunc.bErr THEN
		fbConfirmMFunc(bExecute:= FALSE, sNciToPlc:= sNciToPlc, sPlcToNci:= sPlcToNci);
		bConfirmMFunc	:= FALSE;
		bError		:= TRUE;
		nErrorId	:= fbStepOnAfterEStop.nErrId;
		nState		:= 9000;
	END_IF
	
320:
	(* Reset Channel	*)
	fbNciReset(
		bExecute	:= TRUE, 
		tTimeOut	:= T#500MS, 
		sNciToPlc	:= sNciToPLC );
		
	IF NOT fbNciReset.bBusy AND NOT fbNciReset.bErr THEN
		fbNciReset(bExecute := FALSE, sNciToPlc := sNciToPLC);
		nState		:= 40;
		nLastState	:= nState;
	ELSIF fbNciReset.bErr THEN
		fbNciReset(bExecute := FALSE, sNciToPlc := sNciToPLC);
		bError		:= TRUE;
		nErrorId	:= fbNciReset.nErrId;
		nState		:= 9000;
	END_IF
	
400:
	(* Clear group	*)
	fbClearGroup(
		bExecute	:= TRUE, 
		nGroupId	:= ItpGetGroupId(sNciToPlc:= sNciToPlc), 
		tTimeOut	:= T#200MS);
		
	IF NOT fbClearGroup.bBusy AND NOT fbClearGroup.bErr THEN
		fbClearGroup(bExecute := FALSE);
		bBuildGroupDone	:= FALSE;
		nState		:= 410;
		nLastState	:= nState;
	ELSIF fbClearGroup.bErr THEN
		fbClearGroup(bExecute := FALSE);
		bError		:= TRUE;
		nErrorId	:= fbClearGroup.nErrId;
		nState		:= 9000;
	END_IF 
	
410:
	(* Check for not enable and not start	*)
	IF (NOT bEnable) AND (NOT bStart) THEN
		nState		:= 0;
		nLastState	:= nState;
	END_IF
	
	
9000:
	(* Error happened	*)
	IF (NOT bEnable) AND (NOT bStart) THEN
		IF bBuildGroupDone THEN
			nState		:= 9010;
			nLastState	:= nState;
		ELSE
			nState		:= 0;
			nLastState	:= nState;
		END_IF
	END_IF
	
9010:
	 (* Clear group	*)
	fbClearGroup(
		bExecute	:= TRUE, 
		nGroupId	:= ItpGetGroupId(sNciToPlc:= sNciToPlc), 
		tTimeOut	:= T#200MS);
		
	IF NOT fbClearGroup.bBusy AND NOT fbClearGroup.bErr THEN
		fbClearGroup(bExecute := FALSE);
		bBuildGroupDone	:= FALSE;
		nState		:= 0;
		nLastState	:= nState;
	ELSIF fbBuildGroup.bErr THEN
		fbClearGroup(bExecute := FALSE);
		bError		:= TRUE;
		nErrorId	:= fbClearGroup.nErrId;
		nState		:= 9000;
	END_IF 
	
END_CASE

END_FUNCTION_BLOCK

// ---- POUs/NCI/FB_NciWriteToolParams.TcPOU
FUNCTION_BLOCK FB_NciWriteToolParams
VAR_INPUT
	bExecute			: BOOL;
END_VAR
VAR_IN_OUT
	sNciToPLC			: NCTOPLC_NCICHANNEL_REF;
END_VAR
VAR_OUTPUT
	bDone				: BOOL;
	bBusy				: BOOL;
	bError				: BOOL;
	nErrorId			: UDINT;
END_VAR
VAR
	fbWriteToolDesc		: ItpWriteToolDescEx;
	nState				: INT;
	nLastState			: INT;
	nToolIndex			: UDINT;
END_VAR


CASE nState OF

0:
	bDone		:= FALSE;
	bBusy		:= FALSE;
	bError		:= FALSE;
	nErrorId	:= 0;

	IF bExecute THEN
		nToolIndex	:= 1;
		bBusy		:= TRUE;
		nState		:= 10;
		nLastState	:= nState;
	END_IF	
	
10:
	fbWriteToolDesc(
		bExecute	:= TRUE, 
		nDNo		:= nToolIndex, 
		tTimeOut	:= T#200MS, 
		sNciToPlc	:= sNciToPLC, 
		sToolDesc	:= stNciToolParams[nToolIndex]);
		
	IF NOT fbWriteToolDesc.bBusy AND NOT fbWriteToolDesc.bErr THEN
		fbWriteToolDesc( bExecute := FALSE, sNciToPlc := sNciToPLC, sToolDesc := stNciToolParams[nToolIndex] ); 
		nState		:= 20;
		nLastState	:= nState;
	ELSIF fbWriteToolDesc.bErr THEN
		fbWriteToolDesc( bExecute := FALSE, sNciToPlc := sNciToPLC, sToolDesc := stNciToolParams[nToolIndex] ); 
		bError		:= TRUE;
		nErrorId	:= fbWriteToolDesc.nErrId;
		nState		:= 900;
	END_IF
	
20:
	fbWriteToolDesc( bExecute := FALSE, sNciToPlc := sNciToPLC, sToolDesc := stNciToolParams[nToolIndex] );
	
	IF UDINT_TO_DINT(nToolIndex) < cnMaxToolNumber THEN
		nToolIndex	:= nToolIndex + 1;
		nState		:= 10;
		nLastState	:= nState;
	ELSE 
		nState		:= 30;
		nLastState	:= nState;
	END_IF
	
30:
	bBusy	:= FALSE;
	bDone	:= TRUE;
	
	IF NOT bExecute THEN
		nState		:= 0;
		nLastState	:= nState;
	END_IF
	
900:
	bBusy	:= FALSE;
	bDone	:= FALSE;
	
	IF NOT bExecute THEN
		nState		:= 0;
		nLastState	:= nState;
	END_IF

END_CASE

END_FUNCTION_BLOCK

// ---- POUs/NCI/FB_NciMFunctions.TcPOU
FUNCTION_BLOCK FB_NciMFunctions
VAR_IN_OUT
	sNciToPlc		: NCTOPLC_NCICHANNEL_REF;
	sPlcToNci		: PLCTONC_NCICHANNEL_REF;
END_VAR
VAR_OUTPUT
	bBusy			: BOOL;
	bError			: BOOL;
	nErrorId		: UDINT;
END_VAR
VAR
	fbConfirm		: ItpConfirmHsk;
	nAktMfunc		: INT :=  -1;
	bConfirm		: BOOL;
	i				: INT;
END_VAR


(* Check for m function and store information in bMFunc Array	*)
IF ItpIsHskMFunc(sNciToPlc:= sNciToPlc) THEN
	nAktMfunc 			:= ItpGetHskMFunc(sNciToPlc:= sNciToPlc);
	bMFunc[nAktMfunc]	:= TRUE;
ELSE
	nAktMfunc 	:= -1;
	bConfirm 	:= FALSE;
	FOR i := 0 TO cnMaxMFuncNumber DO
		bMFunc[i]		:= FALSE;
		bQuitMFunc[i]	:= FALSE;
	END_FOR
END_IF

(* Confirm M function, if bit in array bQuitMFunc is set *)
IF nAktMfunc <> -1 THEN
	IF bQuitMFunc[nAktMfunc] THEN
		bConfirm	:= TRUE;
	END_IF
	bQuitMFunc[nAktMfunc]	:= FALSE;
END_IF

(* Confirm M function	*)
fbConfirm(
	bExecute	:= bConfirm, 
	sNciToPlc	:= sNciToPlc, 
	sPlcToNci	:= sPlcToNci, 
	bBusy		=> bBusy, 
	bErr		=> bError, 
	nErrId		=> nErrorId);

END_FUNCTION_BLOCK

// ---- POUs/NCI/FB_NciReadLine.TcPOU
FUNCTION_BLOCK FB_NciReadLine
VAR_INPUT
	bEnable			: BOOL;
	tIdleTime		: TIME	:= T#100MS;
END_VAR
VAR_IN_OUT
	sNciToPlc		: NCTOPLC_NCICHANNEL_REF;
END_VAR
VAR_OUTPUT
	sNciLines		: STRING(255);
	sActualLine		: STRING(80);
	bError			: BOOL;
	nErrorId		: UDINT;
END_VAR
VAR
	fbAdsRead		: ADSREADEX;
	fbTimer			: TON;
	sReadString		: STRING(255);
	sTempLine		: STRING(255);
	nState			: INT;
	nNrOfLines		: INT;
	i				: INT;
	nCharPos		: INT;
END_VAR

CASE nState OF

0:
	sReadString	:= '';
	sActualLine	:= '';
	bError		:= FALSE;
	nErrorId	:= 0;
	
	IF bEnable THEN
		nState	:= 10;
	END_IF	
	
10:
	fbAdsRead(
		NETID		:= '', 
		PORT		:= 500, 
		IDXGRP		:= 16#2300 + ItpGetChannelId(sNciToPlc), 
		IDXOFFS		:= 16#2000_0001, 
		LEN			:= SIZEOF(sReadString), 
		DESTADDR	:= ADR(sReadString), 
		READ		:= TRUE, 
		TMOUT		:= T#500MS );
		
	IF NOT fbAdsRead.BUSY AND NOT fbAdsRead.ERR THEN
		fbAdsRead( READ := FALSE);
		nState	:= 20;
	ELSIF fbAdsRead.ERR THEN
		fbAdsRead( READ := FALSE);
		bError		:= TRUE;
		nErrorId	:= fbAdsRead.ERRID;
		nState		:= 900;
	END_IF
	
20:
	nNrOfLines	:= 0;
	sTempLine	:= '';
	sTempLine	:= sReadString;
	sNciLines	:= sReadString;
	
	FOR i:= 1 TO 3 DO
		nCharPos	:= FIND(sTempLine, '$R$N');
		IF nCharPos <> 0 THEN
			sActualLine		:= LEFT(sTempLine, nCharPos-1);
			sTempLine		:= DELETE(STR:=sTempLine , LEN:=nCharPos+1, POS:=1);
			nNrOfLines		:= nNrOfLines + 1;
		ELSE
			EXIT;
		END_IF
	END_FOR
	
	IF NOT bEnable THEN
		nState	:= 0;
	ELSIF tIdleTime = T#0S THEN
		nState	:= 10;
	ELSE
		nState	:= 30;
	END_IF
	
30:
	fbTimer(IN:= TRUE, PT:= tIdleTime );
	IF fbTimer.Q THEN
		fbTimer(IN:= FALSE);
		nState	:= 10;
	END_IF
	
	IF NOT bEnable THEN
		fbTimer(IN:= FALSE);
		nState	:= 0;
	END_IF

900:
	fbTimer(IN:= TRUE, PT:= T#1S );
	IF fbTimer.Q THEN
		fbTimer(IN:= FALSE);
		nState	:= 10;
	END_IF
	
	IF NOT bEnable THEN
		fbTimer(IN:= FALSE);
		nState	:= 0;
	END_IF
	
END_CASE

END_FUNCTION_BLOCK

// ---- POUs/OPC-UA/FB_OpcUAWrite.TcPOU
FUNCTION_BLOCK FB_OpcUAWrite
VAR_INPUT
	bExecute				: BOOL;
	sServerURL				: STRING(MAX_STRING_LENGTH) := 'opc.tcp://tr.kilit.com:4843';
	sNameSpace				: STRING(MAX_STRING_LENGTH)	:= 'urn:CX-27E172:BeckhoffAutomation:Ua:PLC1';
	sNodeNameW				: STRING(MAX_STRING_LENGTH)	:= 'PRG_Delta.arrDataW1';
	sNodeNameR				: STRING(MAX_STRING_LENGTH)	:= 'PRG_Delta.arrDataR1';
	nVariableSizeW			: UINT;
	pVariableAddrW			: PVOID;
	nVariableSizeR			: UINT;
	pVariableAddrR			: PVOID;
	tWaitDataExchange		: TIME :=T#3S;
	tWaitReConnect			: TIME :=T#3S;
END_VAR
VAR_OUTPUT
	bBusy					: BOOL;
	bError					: BOOL;
END_VAR
VAR	
	fbUaConnect				: UA_Connect;
	fbUaGetNamespaceIndex	: UA_GetNamespaceIndex;
	fbUaNodeGetHandle		: UA_NodeGetHandle;
	fbUaWrite				: UA_Write;
	fbUARead				: UA_Read;
	fbUaNodeReleaseHandle	: UA_NodeReleaseHandle;
	fbUaDisconnect			: UA_Disconnect;
	stNodeID				: ST_UANodeID;
	stSessionConnectInfo	: ST_UASessionConnectInfo;
	stNodeAddInfo			: ST_UANodeAdditionalInfo;
	fbWaitSession			: TON;
	fbWaitDataExchange		: TON;
	tWaitDisconnect			: TON;
	arrOpcDataW				: ARRAY[1..420] OF BYTE;
	arrOpcDataR				: ARRAY[1..8] OF BYTE;
	nState					: INT;
	nErrorID				: UDINT;
	nConnectionHdl			: DWORD;
	nNamespaceIndex			: UINT;					
	nNodeHdlW				: DWORD;
	nNodeHdlR				: DWORD;
	tWaitSessionTimeout		: TON;
END_VAR
VAR CONSTANT
	cnMaxConnHandle			: INT	:= 20;
END_VAR


IF nState > 10 AND nState < 80 THEN 
	IF NOT bExecute THEN 
		fbWaitSession(IN:= FALSE);
		fbWaitDataExchange(IN:= FALSE);
		nState 			:= 80;
	END_IF
END_IF



(*OPC UA Writing Sequence*)
CASE nState OF
	
0:
	fbUaConnect									(Execute := FALSE);
	fbUaGetNamespaceIndex						(Execute := FALSE);
	fbUaNodeGetHandle							(Execute := FALSE);
	fbUaWrite									(Execute := FALSE);
	fbUaNodeReleaseHandle						(Execute := FALSE);
	fbUaDisconnect								(Execute := FALSE);
	bBusy										:= FALSE;
	bError										:= FALSE;
	
	stSessionConnectInfo.tConnectTimeout 		:= T#1S;
	stSessionConnectInfo.tSessionTimeout 		:= T#1S;
	stSessionConnectInfo.sApplicationName		:= '';
	stSessionConnectInfo.eSecurityMode 			:= eUASecurityMsgMode_None;
	stSessionConnectInfo.eSecurityPolicyUri 	:= eUASecurityPolicy_None;
	stSessionConnectInfo.eTransportProfileUri 	:= eUATransportProfileUri_UATcp;
	
	IF bExecute THEN
		nState	:= 10;
	END_IF
	
10:
	fbUaConnect(
		Execute				:= TRUE,
		ServerURL			:= sServerURL,
		SessionConnectInfo	:= stSessionConnectInfo,
		Timeout				:= T#5S );
				
	IF NOT fbUaConnect.Busy THEN
		fbUaConnect(Execute := FALSE);
		IF NOT fbUaConnect.Error THEN
			(* session open *)
			nConnectionHdl	:= fbUaConnect.ConnectionHdl;
			bBusy 			:=TRUE;
			nState			:= 30;
		ELSE
			bError			:= TRUE;
			nErrorID		:= fbUaConnect.ErrorID;
			nState			:= 20;
		END_IF
	END_IF
	
20:
	fbUaConnect			(Execute := FALSE);
	fbWaitSession		(IN:= TRUE, PT:= tWaitReConnect);
	IF fbWaitSession.Q THEN
		fbWaitSession	(IN:= FALSE);
		nState 			:= 10;
	END_IF
	
30:
	fbUaGetNamespaceIndex(
		Execute			:= TRUE,
		ConnectionHdl	:= nConnectionHdl,
		NamespaceUri	:= sNameSpace,
		NamespaceIndex	=> nNamespaceIndex );

	IF NOT fbUaGetNamespaceIndex.Busy THEN
		fbUaGetNamespaceIndex(Execute := FALSE);

		IF NOT fbUaGetNamespaceIndex.Error THEN
			nState 		:= 40;
		ELSE
			bError		:= TRUE;
			nErrorID	:= fbUaGetNamespaceIndex.ErrorID;
			nState 		:= 100;
		END_IF
	END_IF
	
40:
	stNodeID.eIdentifierType 	:= eUAIdentifierType_String;
	stNodeID.nNamespaceIndex 	:= nNamespaceIndex;
	stNodeID.sIdentifier		:= sNodeNameW;
	
	fbUaNodeGetHandle(
		Execute					:= TRUE,
		ConnectionHdl			:= nConnectionHdl,
		NodeID					:= stNodeID,
		NodeHdl					=> nNodeHdlW);

	IF NOT fbUaNodeGetHandle.Busy THEN
		fbUaNodeGetHandle(Execute := FALSE);

		IF NOT fbUaNodeGetHandle.Error THEN
			bError				:= FALSE;
			nState				:= 45;
		ELSE
			bError				:= TRUE;
			nErrorID			:= fbUaNodeGetHandle.ErrorID;
			IF nConnectionHdl <>0 THEN 
				nState 			:= 70; (* Connection is Lost. Wait and try again later *)
			ELSE
				nState 			:= 100; (* idle *)
			END_IF
		END_IF
	END_IF
	
45:
	stNodeID.eIdentifierType 	:= eUAIdentifierType_String;
	stNodeID.nNamespaceIndex 	:= nNamespaceIndex;
	stNodeID.sIdentifier		:= sNodeNameR;
	
	fbUaNodeGetHandle(
		Execute					:= TRUE,
		ConnectionHdl			:= nConnectionHdl,
		NodeID					:= stNodeID,
		NodeHdl					=> nNodeHdlR);

	IF NOT fbUaNodeGetHandle.Busy THEN
		fbUaNodeGetHandle(Execute := FALSE);

		IF NOT fbUaNodeGetHandle.Error THEN
			bError				:= FALSE;
			nState				:= 50;
		ELSE
			bError				:= TRUE;
			nErrorID			:= fbUaNodeGetHandle.ErrorID;
			IF nConnectionHdl <>0 THEN 
				nState 			:= 70; (* Connection is Lost. Wait and try again later *)
			ELSE
				nState 			:= 100; (* idle *)
			END_IF
		END_IF
	END_IF
	
50:
	MEMCPY(ADR(arrOpcDataW) , pVariableAddrW , nVariableSizeW);
	nState	:= 51;
	
51:
	fbUaWrite(
		Execute			:= TRUE,
		ConnectionHdl	:= nConnectionHdl,
		NodeHdl			:= nNodeHdlW,
		stNodeAddInfo	:= stNodeAddInfo,
		cbData			:= SIZEOF(arrOpcDataW),
		pVariable		:= ADR(arrOpcDataW) );

	IF NOT fbUaWrite.Busy THEN
		fbUaWrite(
			Execute 	:= FALSE,
			pVariable	:= ADR(arrOpcDataW));

		IF NOT fbUaWrite.Error THEN
			bError		:= FALSE;
			nState 		:= 55; //cyclic writing sequence
		ELSE
			bError		:= TRUE;
			nErrorID	:= fbUaWrite.ErrorID;
			nState 		:= 70; //if Connection is gone ,wait and try again later 
		END_IF
	END_IF
	
55:
	fbUaRead(
		Execute			:= TRUE,
		ConnectionHdl	:= nConnectionHdl,
		NodeHdl			:= nNodeHdlR,
		stNodeAddInfo	:= stNodeAddInfo,
		cbData			:= SIZEOF(arrOpcDataR),
		pVariable		:= ADR(arrOpcDataR) );

	IF NOT fbUaRead.Busy THEN
		fbUaRead(
			Execute 	:= FALSE,
			pVariable	:= ADR(arrOpcDataR));

		IF NOT fbUaRead.Error THEN
			bError		:= FALSE;
			nState 		:= 56; //cyclic writing sequence
		ELSE
			bError		:= TRUE;
			nErrorID	:= fbUaRead.ErrorID;
			nState 		:= 70; //if Connection is gone ,wait and try again later 
		END_IF
	END_IF
	
56:
	MEMCPY(pVariableAddrR , ADR(arrOpcDataR) , nVariableSizeR);
	nState	:= 60;
	
60:
	fbWaitDataExchange(IN:= TRUE, PT:= tWaitDataExchange);
	IF fbWaitDataExchange.Q THEN
		fbWaitDataExchange	(IN:= FALSE);
		nState 				:= 50;
	END_IF

70:
	fbWaitSession(IN:= TRUE, PT:= tWaitReConnect);
	IF fbWaitSession.Q THEN
		fbWaitSession(IN:= FALSE);
		nState 				:= 40;
	END_IF
	
80:
	fbUaNodeReleaseHandle(
		Execute				:= TRUE,
		ConnectionHdl		:= nConnectionHdl,
		NodeHdl				:= nNodeHdlW );

	IF NOT fbUaNodeReleaseHandle.Busy THEN
		fbUaNodeReleaseHandle(Execute := FALSE);

		IF NOT fbUaNodeReleaseHandle.Error THEN
			nState 			:= 81;
		ELSE
			bError			:= TRUE;
			fbUaNodeReleaseHandle(Execute := FALSE);
			nErrorID		:= fbUaNodeReleaseHandle.ErrorID;
			nState 			:= 110; (* idle *)
		END_IF
	END_IF
	
81:
	fbUaNodeReleaseHandle(
		Execute				:= TRUE,
		ConnectionHdl		:= nConnectionHdl,
		NodeHdl				:= nNodeHdlR );

	IF NOT fbUaNodeReleaseHandle.Busy THEN
		fbUaNodeReleaseHandle(Execute := FALSE);

		IF NOT fbUaNodeReleaseHandle.Error THEN
			nState 			:= 100;
		ELSE
			bError			:= TRUE;
			fbUaNodeReleaseHandle(Execute := FALSE);
			nErrorID		:= fbUaNodeReleaseHandle.ErrorID;
			nState 			:= 110; (* idle *)
		END_IF
	END_IF
	
100:
	fbUaDisconnect(
		Execute				:= TRUE,
		Timeout 			:= T#15S,
		ConnectionHdl		:= nConnectionHdl );

	IF NOT fbUaDisconnect.Busy THEN
		fbUaDisconnect(Execute:= FALSE,ConnectionHdl:= nConnectionHdl );
		IF NOT fbUaDisconnect.Error THEN
			(* session closed *)
			nConnectionHdl	:= 0;
			bBusy 			:= FALSE; 
			nState 			:= 0;
			IF NOT bError THEN 
				bBusy 		:= FALSE;
			END_IF
		ELSE
			//if session handle was invalid 
			nConnectionHdl	:= 0;
			bBusy 			:= FALSE; 
			nState 			:= 110;
		END_IF
	END_IF
	
110:
	tWaitSessionTimeout(IN := TRUE, PT := (tWaitReConnect) );
	IF tWaitSessionTimeout.Q THEN 
		tWaitSessionTimeout(IN :=FALSE);
		nState := 0;
	END_IF
	
END_CASE

END_FUNCTION_BLOCK

// ---- POUs/OPC-UA/PRG_OpcUA.TcPOU
PROGRAM PRG_OpcUA
VAR
	//OPC UA Variables
	fbOpcUAWrite	: FB_OpcUAWrite;
	tStartComm		: TON;
	nTest			: INT;
	bExecute		: BOOL;
	bBusy			: BOOL;
	bError			: BOOL;
END_VAR

//OPC UA 
(*Servera gönderilecek bilgiler*)

tStartComm(IN:= NOT bExecute, PT:= T#5S);
IF  tStartComm.Q THEN 
	bExecute	:= TRUE;
END_IF

fbOpcUAWrite(
	bExecute			:= bExecute,
	sServerURL			:= 'opc.tcp://tr.kilit.com:4843',	
	sNameSpace			:= 'urn:KILIT-C01:BeckhoffAutomation:Ua:PLC1',
	sNodeNameW			:='PRG_Delta.arrDataW1', 
	sNodeNameR			:='PRG_Delta.arrDataR1',
	nVariableSizeW		:= SIZEOF(GVL_Process.stOpcUaVariablesW),
	pVariableAddrW		:= ADR(GVL_Process.stOpcUaVariablesW),
	nVariableSizeR		:= SIZEOF(GVL_Process.stOpcUaVariablesR),
	pVariableAddrR		:= ADR(GVL_Process.stOpcUaVariablesR),
	tWaitDataExchange	:=T#1S , 
	tWaitReConnect		:=T#4S ,
	bBusy				=>bBusy , 
	bError				=>bError );

END_PROGRAM

// ---- POUs/PRG_MFuncControl.TcPOU
PROGRAM PRG_MFuncControl
VAR
	bTestValveOutput		: BOOL;
END_VAR


IF bMFunc[11] THEN
	bTestValveOutput	:= TRUE;
	bQuitMFunc[11]		:= TRUE;
END_IF


IF bMFunc[12] THEN
	bTestValveOutput	:= FALSE;
	bQuitMFunc[12]		:= TRUE;
END_IF

END_PROGRAM

// ---- POUs/PRG_Process.TcPOU
PROGRAM PRG_Process
VAR
	bTempAllAxisEnable		: BOOL;	
	bTempAllAxisReset		: BOOL;	
	bTempAllAxisEnableHMI	: BOOL;
	bInvisible				: BOOL := TRUE;
	bMode					: BOOL;
	bAutoMode				: BOOL;
	bManualMode				: BOOL;
	nStateEnable			: INT;
		
	nStateReset				: INT;
	nStateFrame				: INT;
	
	nStateAutoMan			: INT;
	nLastStateAutoMan		: INT;
	tWaitEnable				: TON;
	tWaitNciGroupDone		: TON;
	
	nStatePathChange		: INT;
	
	fbFindFileList			: FB_EnumFindFileList ;
	   	sNetID     			: T_AmsNetID 	:= '';
    	sPathName  			: T_MaxString 	:= 'C:\TwinCAT\CNC\*.nc';
		arrFileList			: ARRAY[0..20] OF ST_FindFileEntry;
   		bExecuteFindList	: BOOL;
  
	i						: INT;
	arrFileNameList			: ARRAY[0..20] OF STRING;
	nFileNameList			: INT;
	nLastFileNameList		: INT;
	nStateFileNameList		: INT;
	bChangeFile				: BOOL;
	bSelectFile				: BOOL;
	bCancelSelectFile		: BOOL;
	//Delta içerisindeki G codelarına göre degistirilecek
	sFileName				: STRING := 'C:\TwinCAT\CNC\Beckhoff_Robot_Yatirimlari_2.NC';
	sFileNameVisu			: STRING := 'Beckhoff_Robot_Yatirimlari_2.NC';
	tUpdatePathList			: TON;		
	
	//Otomatik HMI Acılsın
	ntStartHMI				: NT_StartProcess;
	tTimerStartHMI			: TON;
	
	// Windows XP ve üzeri isletim sistemleri icin kullanilan FB
	fbScreenOff		: FB_ScreenOnOff_Win7;
		bScreenOff	: BOOL;
		bDone		: BOOL;
	tTimerScreenOff	: TON;
		bOff		: BOOL;
		
	//Enable PLC or HMI 
	nStateEnableHP	: INT;
	nStateNciHP		: INT;
END_VAR

ACT_EnableReset();
ACT_NciPathChange();
ACT_AxisSelectOnManualMode();
ACT_AutoManualMode();
ACT_FromTC3toTwinCATHMI();




tTimerStartHMI(IN:= TRUE, PT:= T#10S);

IF tTimerStartHMI.Q THEN 

ntStartHMI(
	NETID		:= , 
	PATHSTR		:= 'C:\TwinCAT\3.1\Components\Plc\Tc3PlcHmi\Tc3PlcHmi.exe', 
	DIRNAME		:= 'C:\TwinCAT\3.1\Components\Plc\Tc3PlcHmi', 
	COMNDLINE	:= , 
	START		:= TRUE, 
	TMOUT		:= T#5S, 
	BUSY		=> , 
	ERR			=> , 
	ERRID		=> );
END_IF 

tTimerScreenOff(IN:= bOff, PT:= T#5S);

IF tTimerScreenOff.Q THEN 
	bScreenOff	:= TRUE;
	IF bDone THEN 
		bScreenOff	:= FALSE;
		bOff		:= FALSE;
	END_IF
END_IF

fbScreenOff(
	bScreenOff	:= bScreenOff , 
	bDone		=> bDone );

ACTION ACT_AutoManualMode:
//Otomatic-Manual Modelar arasındaki geçişlerde değişkenlerin ayarlanmasi
IF VisuElems.CURRENTVISU = 'Visualization_AxesInfo_Manual' THEN 
	GVL_Process.nAutoManMode	:= FALSE;
ELSIF VisuElems.CURRENTVISU = 'Visualization_AxesInfo' THEN 
	GVL_Process.nAutoManMode	:= TRUE;
END_IF 

CASE nStateAutoMan OF 
0:	
	IF GVL_Process.nAutoManMode THEN 
		nLastStateAutoMan	:= nStateAutoMan;
		nStateAutoMan		:= 50;
	ELSE
		nLastStateAutoMan	:= nStateAutoMan;
		nStateAutoMan		:= 150;
	END_IF
	
50:
	IF (NOT stAxisM1_B.Out.xAxisError) AND 
		(NOT stAxisM2_C.Out.xAxisError) AND 
		(NOT stAxisM3_A.Out.xAxisError) AND 
		(NOT stAxisX.Out.xAxisError) AND 
		(NOT stAxisY.Out.xAxisError) AND 
		(NOT stAxisZ.Out.xAxisError) AND 
		(NOT stAxisM2_C.Out.xAxisError) AND
		(NOT stAxisM1_B.Out.xDriveError) AND 
 		(NOT stAxisM2_C.Out.xDriveError) AND
		(NOT stAxisM3_A.Out.xDriveError) AND
		(NOT stAxisX.Out.xDriveError) AND
		(NOT stAxisY.Out.xDriveError) AND
		(NOT stAxisZ.Out.xDriveError) THEN 
		nStateAutoMan		:= 60;
	ELSE
		//Error Durumunda Reset State ine gönderilecek
		nLastStateAutoMan	:= nStateAutoMan;
		nStateAutoMan		:= 900;
	END_IF 

60:
	GVL_Process.bAllAxesEnablePLC	:= TRUE;//GVL_Process.bAllAxesEnable 	:= TRUE;
	tWaitEnable(IN:= TRUE, PT:= T#250MS);
	IF tWaitEnable.Q THEN 
		tWaitEnable(IN:= FALSE);
		nStateAutoMan	:= 65;
	END_IF

65:
	IF stAxisM1_B.Out.xEnabled AND 
		stAxisM2_C.Out.xEnabled AND 
		stAxisM3_A.Out.xEnabled AND 
		stAxisX.Out.xEnabled AND 
		stAxisY.Out.xEnabled AND 
		stAxisZ.Out.xEnabled THEN 
		PRG_Kinematic.bExecuteKinConfigGroup	:=FALSE;
		nStateAutoMan	:= 70;
	ELSE
	 	//Error Durumunda Reset State ine gönderilecek
		nLastStateAutoMan	:= nStateAutoMan;
		nStateAutoMan		:= 900;
	END_IF
	
70:
	IF NOT PRG_Kinematic.fbKinConfigGroup.bError THEN 
		PRG_Kinematic.bCartesianMode			:= TRUE;
		PRG_Kinematic.bExecuteKinConfigGroup	:= TRUE;
		IF PRG_Kinematic.fbKinConfigGroup.bDone THEN
			PRG_Kinematic.bExecuteKinConfigGroup	:= FALSE; 
			nStateAutoMan	:= 80;
		END_IF
	ELSE
		//Error Durumunda Reset State ine gönderilecek
		nLastStateAutoMan	:= nStateAutoMan;
		nStateAutoMan		:= 900;
	END_IF

80:
	tWaitNciGroupDone(IN:= TRUE, PT:= T#1S);
	IF NOT PRG_NcControl.bNciError THEN 
		PRG_NcControl.bNciEnable	:= TRUE;
		IF PRG_NcControl.bBuildGroupDone THEN 
			nStateAutoMan	:= 90;
		ELSIF tWaitNciGroupDone.Q THEN 				//KONTROL ET
			tWaitNciGroupDone(IN:= FALSE); 
			PRG_NcControl.bNciEnable	:= FALSE;
			nStateAutoMan	:= 0;
		END_IF
	ELSE 
		//Error Durumunda Reset State ine gönderilecek
		nLastStateAutoMan	:= nStateAutoMan;
		nStateAutoMan		:= 900;
	END_IF
	
90:
	//Auto Mode Dan manual a geçme
	IF NOT GVL_Process.nAutoManMode THEN 
		IF PRG_NcControl.bProgramRunning 
			AND NOT PRG_NcControl.bProgramStopped
			AND NOT PRG_NcControl.bProgramFinished THEN 
				PRG_NcControl.bNciStart		:= FALSE; //GVL_Process.bNciStartPLC	:= FALSE; 		
		END_IF
		nStateAutoMan				:= 100;	
	END_IF

100:
	IF NOT PRG_NcControl.bNciError THEN 
		nStateAutoMan	:= 110;
	ELSE
		//Error Durumunda Reset State ine gönderilecek
		nLastStateAutoMan	:= nStateAutoMan;
		nStateAutoMan		:= 900;
	END_IF
	
110:
	IF NOT PRG_NcControl.bProgramRunning 
		OR PRG_NcControl.bProgramStopped THEN 
		PRG_NcControl.bNciStart		:= FALSE; //GVL_Process.bNciStartPLC	:= FALSE; 
		PRG_NcControl.bNciEnable	:= FALSE;
		nStateAutoMan				:= 150;
	END_IF
		
150:
	IF (NOT stAxisM1_B.Out.xAxisError) AND 
		(NOT stAxisM2_C.Out.xAxisError) AND 
		(NOT stAxisM3_A.Out.xAxisError) AND 
		(NOT stAxisX.Out.xAxisError) AND 
		(NOT stAxisY.Out.xAxisError) AND 
		(NOT stAxisZ.Out.xAxisError) AND 
		(NOT stAxisM2_C.Out.xAxisError) AND
		(NOT stAxisM1_B.Out.xDriveError) AND 
 		(NOT stAxisM2_C.Out.xDriveError) AND
		(NOT stAxisM3_A.Out.xDriveError) AND
		(NOT stAxisX.Out.xDriveError) AND
		(NOT stAxisY.Out.xDriveError) AND
		(NOT stAxisZ.Out.xDriveError) THEN 
		nStateAutoMan		:= 160;
	ELSE
		//Error Durumunda Reset State ine gönderilecek
		nLastStateAutoMan	:= nStateAutoMan;
		nStateAutoMan		:= 900;
	END_IF 	

160:
	GVL_Process.bAllAxesEnablePLC	:= TRUE; //GVL_Process.bAllAxesEnable	:= TRUE;
	tWaitEnable(IN:= TRUE, PT:= t#250ms);
	IF tWaitEnable.Q THEN 
		tWaitEnable(IN:= FALSE);
		nStateAutoMan	:= 165;
	END_IF

165:
	IF stAxisM1_B.Out.xEnabled AND 
		stAxisM2_C.Out.xEnabled AND 
		stAxisM3_A.Out.xEnabled AND 
		stAxisX.Out.xEnabled AND 
		stAxisY.Out.xEnabled AND 
		stAxisZ.Out.xEnabled THEN 
		PRG_Kinematic.bExecuteKinConfigGroup	:=FALSE;
		nStateAutoMan	:= 170;
	ELSE
	 	//Error Durumunda Reset State ine gönderilecek
		nLastStateAutoMan	:= nStateAutoMan;
		nStateAutoMan		:= 900;
	END_IF
	
170:
	IF NOT PRG_Kinematic.fbKinConfigGroup.bError THEN 
		PRG_Kinematic.bCartesianMode			:= TRUE;
		PRG_Kinematic.bExecuteKinConfigGroup	:= TRUE;
		IF PRG_Kinematic.fbKinConfigGroup.bDone THEN 
			PRG_Kinematic.bExecuteKinConfigGroup	:= FALSE;
			nStateAutoMan							:= 180;
		END_IF
	ELSE
		//Error Durumunda Reset State ine gönderilecek
		nLastStateAutoMan	:= nStateAutoMan;
		nStateAutoMan		:= 900;
	END_IF
	
180:
	//Manual dan Auto ya geçme
	IF GVL_Process.nAutoManMode THEN 
		nStateAutoMan	:= 50;
	END_IF
	
900:
//Error State
	IF (NOT stAxisM1_B.Out.xAxisError) AND 
		(NOT stAxisM2_C.Out.xAxisError) AND 
		(NOT stAxisM3_A.Out.xAxisError) AND 
		(NOT stAxisX.Out.xAxisError) AND 
		(NOT stAxisY.Out.xAxisError) AND 
		(NOT stAxisZ.Out.xAxisError) AND 
		(NOT stAxisM2_C.Out.xAxisError) AND
		(NOT stAxisM1_B.Out.xDriveError) AND 
 		(NOT stAxisM2_C.Out.xDriveError) AND
		(NOT stAxisM3_A.Out.xDriveError) AND
		(NOT stAxisX.Out.xDriveError) AND
		(NOT stAxisY.Out.xDriveError) AND
		(NOT stAxisZ.Out.xDriveError) THEN 
		nStateAutoMan	:= 910;
	END_IF 

910:
	IF PRG_Kinematic.fbKinConfigGroup.bError THEN 
		PRG_Kinematic.bExecuteKinResetGroup	:= TRUE;
		nStateAutoMan						:= 920;
	ELSE
		nStateAutoMan						:= 950;
	END_IF
	
920:
	IF PRG_Kinematic.fbKinConfigGroup.bError THEN 
		PRG_Kinematic.bExecuteKinResetGroup	:= FALSE;
		nStateAutoMan						:= 950;
	END_IF
	
950:
	IF GVL_Process.nAutoManMode THEN 
		nStateAutoMan	:= 50;
	ELSE
		nStateAutoMan	:= 150;
	END_IF

END_CASE
END_ACTION

ACTION ACT_AxisSelectOnManualMode:
//HMI da Manual Ekrandan Eksen Seçimi Adimlari
IF NOT GVL_Process.bManualSelectX
	AND NOT GVL_Process.bManualSelectY
	AND NOT GVL_Process.bManualSelectZ THEN 
		GVL_Process.bManualSelectX	:= TRUE;
END_IF

CASE nStateFrame OF 

0:
	GVL_Process.bManualSelectY	:= FALSE;
	GVL_Process.bManualSelectZ	:= FALSE;	
	GVL_Process.nSizeSelectX	:= 35;
	GVL_Process.nSizeSelectY	:= 27;
	GVL_Process.nSizeSelectZ	:= 27;
	nStateFrame					:= 5;
5:
	IF GVL_Process.bManualSelectY THEN 
		nStateFrame	:= 10;
	ELSIF GVL_Process.bManualSelectZ THEN 
		nStateFrame	:= 20;
	END_IF
10:
	GVL_Process.bManualSelectX	:= FALSE;
	GVL_Process.bManualSelectZ	:= FALSE;	
	GVL_Process.nSizeSelectX	:= 27;
	GVL_Process.nSizeSelectY	:= 35;
	GVL_Process.nSizeSelectZ	:= 27;
	nStateFrame					:= 15;
15:
	IF GVL_Process.bManualSelectX THEN 
		nStateFrame	:= 0;
	ELSIF GVL_Process.bManualSelectZ THEN 
		nStateFrame	:= 20;
	END_IF
20:
	GVL_Process.bManualSelectX	:= FALSE;
	GVL_Process.bManualSelectY	:= FALSE;	
	GVL_Process.nSizeSelectX	:= 27;
	GVL_Process.nSizeSelectY	:= 27;
	GVL_Process.nSizeSelectZ	:= 35;
	nStateFrame					:= 25;
25:
	IF GVL_Process.bManualSelectX THEN 
		nStateFrame	:= 0;
	ELSIF GVL_Process.bManualSelectY THEN 
		nStateFrame	:= 10;
	END_IF

END_CASE
END_ACTION

ACTION ACT_EnableReset:
//All Axes Enable 
// bTemp.. degiskeni bir kerelik enable kesme isleminde kullanıldı
(*IF bTempAllAxisEnable AND NOT GVL_Process.bAllAxesEnable THEN 
	nStateEnable	:= 0;
END_IF*)

CASE nStateEnable OF 
0:
	IF GVL_Process.bAllAxesEnable THEN 
		stAxisX.In.xEnable		:= TRUE;
		stAxisY.In.xEnable		:= TRUE;
		stAxisZ.In.xEnable		:= TRUE;
		stAxisM1_B.In.xEnable	:= TRUE;
		stAxisM2_C.In.xEnable	:= TRUE;
		stAxisM3_A.In.xEnable	:= TRUE;
		bTempAllAxisEnable		:= TRUE;
		bTempAllAxisEnableHMI	:= TRUE;
		nStateEnable			:= 10;
	ELSIF bTempAllAxisEnable AND NOT GVL_Process.bAllAxesEnable THEN 
		stAxisX.In.xEnable		:= FALSE;
		stAxisY.In.xEnable		:= FALSE;
		stAxisZ.In.xEnable		:= FALSE;
		stAxisM1_B.In.xEnable	:= FALSE;
		stAxisM2_C.In.xEnable	:= FALSE;
		stAxisM3_A.In.xEnable	:= FALSE;
		bTempAllAxisEnableHMI	:= FALSE;
		bTempAllAxisEnable		:= FALSE;
(*	ELSIF bTempAllAxisEnableHMI OR GVL_Process.stOpcUaVariablesR.bEnableAllProcess THEN
		stAxisX.In.xEnable		:= FALSE;
		stAxisY.In.xEnable		:= FALSE;
		stAxisZ.In.xEnable		:= FALSE;
		stAxisM1_B.In.xEnable	:= FALSE;
		stAxisM2_C.In.xEnable	:= FALSE;
		stAxisM3_A.In.xEnable	:= FALSE;
		bTempAllAxisEnableHMI	:= FALSE;
		bTempAllAxisEnable		:= FALSE;*)
	END_IF
	
10:
	IF NOT PRG_Kinematic.fbKinConfigGroup.bError THEN 
		PRG_Kinematic.bExecuteKinResetGroup		:= FALSE;
		PRG_Kinematic.bExecuteKinConfigGroup 	:= TRUE;
		nStateEnable	:= 20;
	ELSE
		PRG_Kinematic.bExecuteKinResetGroup	:= TRUE;
	END_IF 
	
20:
	IF VisuElems.CURRENTVISU = 'Visualization_AxesInfo_Manual' THEN 
		nStateEnable	:= 50;
	ELSIF VisuElems.CURRENTVISU = 'Visualization_AxesInfo' THEN
		nStateEnable	:= 150;
	END_IF

50:
	IF NOT GVL_Process.bAllAxesEnable THEN 
		nStateEnable	:= 170;
	END_IF
	
150:
	IF NOT PRG_NcControl.bNciError THEN 
		PRG_NcControl.bNciEnable	:= TRUE;
		nStateEnable				:= 160;
	END_IF

160:
	IF NOT GVL_Process.bAllAxesEnable THEN 
		nStateEnable	:= 170;
	END_IF
	
170:
	GVL_Process.bAllAxesReset	:= TRUE;
	IF nStateReset = 60 THEN 
		GVL_Process.bAllAxesReset	:= FALSE;
		nStateEnable	:= 180;
	END_IF
	
180:
	GVL_Process.bAllAxesReset	:= TRUE;
	IF nStateReset = 60 THEN 
		GVL_Process.bAllAxesReset	:= FALSE;
		nStateEnable	:= 0;
	END_IF
	
END_CASE



//Kinematic ile otomatik 'Cartesian mode' Active-Inactive
IF nStateReset = 0 THEN 
	IF GVL_Kin.stKinToPLC.ChnOperationState = 4 THEN 
		PRG_Kinematic.bCartesianMode	:= FALSE;
	ELSIF GVL_Kin.stKinToPLC.ChnOperationState = 0 THEN 
		PRG_Kinematic.bCartesianMode	:= FALSE;
	ELSIF GVL_Kin.stKinToPLC.ChnOperationState = 1 THEN 
		PRG_Kinematic.bCartesianMode	:= TRUE;
	END_IF
END_IF 

CASE nStateReset OF  
0: 
	IF GVL_Process.bAllAxesReset THEN
		nStateReset	:= 10;
	END_IF

10:
	//NCI Start Reset
	IF PRG_NcControl.bNciStart THEN  //GVL_Process.bNciStartPLC	THEN  
		PRG_NcControl.bNciStart	:= FALSE;  //GVL_Process.bNciStartPLC	:= FALSE; 
		nStateReset	:= 20;
	ELSE
		nStateReset	:= 20;
	END_IF
	
20:
	//NCI Enable Reset
	IF PRG_NcControl.bNciEnable THEN 
		PRG_NcControl.bNciEnable	:= FALSE;
		nStateReset	:= 30;
	ELSE
		nStateReset	:= 30;
	END_IF

30:
	//Kinematic Cartesian Mode Reset
	IF PRG_Kinematic.bCartesianMode THEN 
		PRG_Kinematic.bCartesianMode	:= FALSE;
	ELSE
		PRG_Kinematic.bExecuteKinConfigGroup := TRUE;
		nStateReset	:= 40;
	END_IF
	
40:
	// Kinematic Reset
	IF NOT PRG_Kinematic.fbKinConfigGroup.bError THEN 
		PRG_Kinematic.bExecuteKinConfigGroup := FALSE;
		nStateReset	:= 50;
	END_IF 
	
50:
	//Axes Reset
	GVL_Axis.stAxisM1_B.In.xReset	:= TRUE;
	GVL_Axis.stAxisM2_C.In.xReset	:= TRUE;
	GVL_Axis.stAxisM3_A.In.xReset	:= TRUE;
	GVL_Axis.stAxisX.In.xReset		:= TRUE;
	GVL_Axis.stAxisY.In.xReset		:= TRUE;
	GVL_Axis.stAxisZ.In.xReset		:= TRUE;
	PRG_Kinematic.bExecuteKinResetGroup	:= TRUE;
	IF NOT GVL_Axis.stAxisM1_B.Out.xAxisError AND NOT GVL_Axis.stAxisM2_C.Out.xAxisError
		AND NOT GVL_Axis.stAxisM3_A.Out.xAxisError AND NOT GVL_Axis.stAxisX.Out.xAxisError
		AND NOT GVL_Axis.stAxisY.Out.xAxisError AND NOT GVL_Axis.stAxisZ.Out.xAxisError THEN 
			GVL_Axis.stAxisM1_B.In.xReset	:= FALSE;
			GVL_Axis.stAxisM2_C.In.xReset	:= FALSE;
			GVL_Axis.stAxisM3_A.In.xReset	:= FALSE;
			GVL_Axis.stAxisX.In.xReset		:= FALSE;
			GVL_Axis.stAxisY.In.xReset		:= FALSE;
			GVL_Axis.stAxisZ.In.xReset		:= FALSE;
			PRG_Kinematic.bExecuteKinResetGroup	:= FALSE;
			nStateReset						:= 60;
	END_IF
	
60:
	PRG_Kinematic.bCartesianMode	:= TRUE;
	IF NOT GVL_Process.bAllAxesReset THEN 
		nStateReset	:= 0;
	END_IF
END_CASE

//Eğer AllAxisEnable Yoksa NCI Starta Basılamasın
IF NOT GVL_Process.bAllAxesEnable THEN 
	PRG_NcControl.bNciStart	:= FALSE; //GVL_Process.bNciStartPLC	:= FALSE; 
END_IF

// Butun eksenler enable oldugunda tek 1 bit aktif olsun 
	IF stAxisM1_B.Out.xEnabled AND 
		stAxisM2_C.Out.xEnabled AND 
		stAxisM3_A.Out.xEnabled AND 
		stAxisX.Out.xEnabled AND 
		stAxisY.Out.xEnabled AND 
		stAxisZ.Out.xEnabled THEN 
			GVL_Process.bAllAxesEnabled	:= TRUE;
	ELSE
			GVL_Process.bAllAxesEnabled	:= FALSE;
	END_IF
END_ACTION

ACTION ACT_FromTC3toTwinCATHMI:
// From TC3 to TwinCAT HMI
	GVL_Process.stOpcUaVariablesW.fActPosX			:= GVL_Axis.AxisX.NcToPlc.ActPos;
	GVL_Process.stOpcUaVariablesW.fActPosY			:= GVL_Axis.AxisY.NcToPlc.ActPos;
	GVL_Process.stOpcUaVariablesW.fActPosZ			:= GVL_Axis.AxisZ.NcToPlc.ActPos;
	GVL_Process.stOpcUaVariablesW.fActPosM1			:= GVL_Axis.AxisM1_B.NcToPlc.ActPos;
	GVL_Process.stOpcUaVariablesW.fActPosM2			:= GVL_Axis.AxisM2_C.NcToPlc.ActPos;
	GVL_Process.stOpcUaVariablesW.fActPosM3			:= GVL_Axis.AxisM3_A.NcToPlc.ActPos;

	GVL_Process.stOpcUaVariablesW.fActVeloX			:= GVL_Axis.AxisX.NcToPlc.SetVelo;
	GVL_Process.stOpcUaVariablesW.fActVeloY			:= GVL_Axis.AxisY.NcToPlc.SetVelo;
	GVL_Process.stOpcUaVariablesW.fActVeloZ			:= GVL_Axis.AxisZ.NcToPlc.SetVelo;
	GVL_Process.stOpcUaVariablesW.fActVeloM1		:= GVL_Axis.AxisM1_B.NcToPlc.SetVelo;
	GVL_Process.stOpcUaVariablesW.fActVeloM2		:= GVL_Axis.AxisM2_C.NcToPlc.SetVelo;
	GVL_Process.stOpcUaVariablesW.fActVeloM3		:= GVL_Axis.AxisM3_A.NcToPlc.SetVelo;
	
	GVL_Process.stOpcUaVariablesW.fLagDistanceX		:= GVL_Axis.AxisX.NcToPlc.PosDiff;	
	GVL_Process.stOpcUaVariablesW.fLagDistanceY		:= GVL_Axis.AxisY.NcToPlc.PosDiff;
	GVL_Process.stOpcUaVariablesW.fLagDistanceZ		:= GVL_Axis.AxisZ.NcToPlc.PosDiff;
	GVL_Process.stOpcUaVariablesW.fLagDistanceM1	:= GVL_Axis.AxisM1_B.NcToPlc.PosDiff;
	GVL_Process.stOpcUaVariablesW.fLagDistanceM2	:= GVL_Axis.AxisM2_C.NcToPlc.PosDiff;
	GVL_Process.stOpcUaVariablesW.fLagDistanceM3	:= GVL_Axis.AxisM3_A.NcToPlc.PosDiff;

	
	GVL_Process.stOpcUaVariablesW.sNciActLine		:= PRG_NcControl.sNciActualLine;
	GVL_Process.stOpcUaVariablesW.sNciLines			:= PRG_NcControl.sNciLines;
	GVL_Process.stOpcUaVariablesW.sFileNameVisu		:= sFileNameVisu;
	
	GVL_Process.stOpcUaVariablesW.bNciRunning		:= PRG_NcControl.bProgramRunning;
	GVL_Process.stOpcUaVariablesW.bNciStopped		:= PRG_NcControl.bProgramStopped;
	GVL_Process.stOpcUaVariablesW.bNciFinished		:= PRG_NcControl.bProgramFinished;	
	
	GVL_Process.stOpcUaVariablesW.bEnabledX			:= GVL_Axis.stAxisX.Out.xEnabled;
	GVL_Process.stOpcUaVariablesW.bEnabledY			:= GVL_Axis.stAxisY.Out.xEnabled;
	GVL_Process.stOpcUaVariablesW.bEnabledZ			:= GVL_Axis.stAxisZ.Out.xEnabled;
	GVL_Process.stOpcUaVariablesW.bEnabledM1		:= GVL_Axis.stAxisM1_B.Out.xEnabled;
	GVL_Process.stOpcUaVariablesW.bEnabledM2		:= GVL_Axis.stAxisM2_C.Out.xEnabled;
	GVL_Process.stOpcUaVariablesW.bEnabledM3		:= GVL_Axis.stAxisM3_A.Out.xEnabled;
	
	GVL_Process.stOpcUaVariablesW.bErrorX			:= GVL_Axis.stAxisX.Out.xAxisError;
	GVL_Process.stOpcUaVariablesW.bErrorY			:= GVL_Axis.stAxisY.Out.xAxisError;
	GVL_Process.stOpcUaVariablesW.bErrorZ			:= GVL_Axis.stAxisZ.Out.xAxisError;
	GVL_Process.stOpcUaVariablesW.bErrorM1			:= GVL_Process.nAutoManMode; //Degistirildi GVL_Axis.stAxisM1_B.Out.xAxisError;
	GVL_Process.stOpcUaVariablesW.bErrorM2			:= GVL_Process.bNciStartPLC; //Degistirildi GVL_Axis.stAxisM2_C.Out.xAxisError;
	GVL_Process.stOpcUaVariablesW.bErrorM3			:= GVL_Process.bAllAxesEnablePLC;	//Değiştirildi GVL_Axis.stAxisM3_C.Out.xAxisError;
	

	
//From TwinCAT HMI to TC3 Enable
CASE nStateEnableHP OF  
0:
	IF NOT GVL_Process.bAllAxesEnable THEN 
		nStateEnableHP	:= 10;
	END_IF
10:
	IF GVL_Process.bAllAxesEnablePLC THEN 
		GVL_Process.bAllAxesEnable	:= TRUE;
		nStateEnableHP	:= 50;
	ELSIF GVL_Process.stOpcUaVariablesR.bEnableAllProcess THEN 
		GVL_Process.bAllAxesEnablePLC	:= TRUE;
		GVL_Process.bAllAxesEnable		:= TRUE;
		nStateEnableHP	:= 100;
	END_IF
	
50:
	IF GVL_Process.stOpcUaVariablesR.bEnableAllProcess THEN 
		nStateEnableHP	:= 150;
	END_IF

100:
	IF GVL_Process.bAllAxesEnablePLC THEN 
		nStateEnableHP	:= 150;
	END_IF  
	
150:
	IF NOT PRG_NcControl.bNciStart THEN 
		IF NOT GVL_Process.bAllAxesEnablePLC  THEN 
			GVL_Process.bAllAxesEnable		:= FALSE;
			nStateEnableHP	:= 200;
		ELSIF NOT GVL_Process.stOpcUaVariablesR.bEnableAllProcess THEN
			GVL_Process.bAllAxesEnablePLC	:= FALSE;
			GVL_Process.bAllAxesEnable		:= FALSE;
			nStateEnableHP	:= 210; 
		END_IF
	ELSIF PRG_NcControl.bNciStart AND NOT GVL_Process.bAllAxesEnablePLC THEN 
		GVL_Process.bAllAxesEnablePLC	:= TRUE;
	END_IF 

200:
	IF NOT GVL_Process.stOpcUaVariablesR.bEnableAllProcess THEN 
		nStateEnableHP	:= 0; 
	END_IF

210:
	IF NOT GVL_Process.bAllAxesEnablePLC THEN 
		nStateEnableHP	:= 0; 
	END_IF
END_CASE


	
//From TwinCAT HMI to TC3 NciStates
IF GVL_Process.nAutoManMode	THEN 
	
	CASE nStateNciHP OF  
	0:
		IF NOT PRG_NcControl.bNciStart THEN 
			nStateNciHP	:= 10;
		END_IF
	10:
		IF GVL_Process.bNciStartPLC THEN 
			PRG_NcControl.bNciStart	:= TRUE;
			nStateNciHP	:= 50;
		ELSIF GVL_Process.stOpcUaVariablesR.bNciStart THEN 
			GVL_Process.bNciStartPLC	:= TRUE;
			PRG_NcControl.bNciStart		:= TRUE;
			nStateNciHP	:= 100;
		END_IF
		
	50:
		IF GVL_Process.stOpcUaVariablesR.bNciStart THEN 
			nStateNciHP	:= 150;
		END_IF
	
	100:
		IF GVL_Process.bNciStartPLC THEN 
			nStateNciHP	:= 150;
		END_IF  
		
	150:
		IF NOT GVL_Process.bNciStartPLC THEN 
			PRG_NcControl.bNciStart		:= FALSE;
			nStateNciHP	:= 200;
		ELSIF NOT GVL_Process.stOpcUaVariablesR.bNciStart THEN
			GVL_Process.bNciStartPLC	:= FALSE;
			PRG_NcControl.bNciStart		:= FALSE;
			nStateNciHP	:= 210; 
		END_IF
	
	200:
		IF NOT GVL_Process.stOpcUaVariablesR.bNciStart
	
	 THEN 
			nStateNciHP	:= 0; 
		END_IF
	
	210:
		IF NOT GVL_Process.bNciStartPLC THEN 
			nStateNciHP	:= 0; 
		END_IF
	END_CASE
	
ELSE
	GVL_Process.bNciStartPLC	:= FALSE;
	nStateNciHP	:= 0;
END_IF 


	//GVL_Process.bAllAxesEnable	:= GVL_Process.stOpcUaVariablesR.bEnableAllProcess;
	//PRG_NcControl.bNciStart		:= GVL_Process.stOpcUaVariablesR.bNciStart;
END_ACTION

ACTION ACT_NciPathChange:
//NCI Path değiştirilirken Kinematic'i Hataya Düşmesin Diye Disable Etme
IF bChangeFile AND (bCancelSelectFile OR bSelectFile) THEN  
	bChangeFile	:= FALSE;
END_IF

CASE nStatePathChange OF 
0:
	IF bChangeFile AND 
		(GVL_Kin.stKinToPLC.ChnOperationState = 4) THEN 
		PRG_Kinematic.bCartesianMode			:= FALSE;
		PRG_Kinematic.bExecuteKinConfigGroup	:= TRUE;
		nStatePathChange						:= 10;
	END_IF
	
10:
	
	IF  (GVL_Kin.stKinToPLC.ChnOperationState = 4) THEN 
		PRG_Kinematic.bExecuteKinConfigGroup	:= FALSE;
		nStatePathChange		:= 15;
	END_IF
	
15:
	IF bChangeFile THEN 
		nStatePathChange	:= 20;
	END_IF 	
	
20:
	IF (NOT bChangeFile) THEN 
		PRG_Kinematic.bExecuteKinConfigGroup	:= TRUE;
		nStatePathChange						:= 30;
	END_IF
	
30:
	IF  (GVL_Kin.stKinToPLC.ChnOperationState = 1) THEN 
		PRG_Kinematic.bExecuteKinConfigGroup	:= FALSE;
		nStatePathChange						:= 40;
	END_IF
	
40:
	PRG_Kinematic.bExecuteKinConfigGroup	:= TRUE;
	IF  (GVL_Kin.stKinToPLC.ChnOperationState = 4) THEN 
		PRG_Kinematic.bExecuteKinConfigGroup	:= FALSE;
		nStatePathChange						:= 0;
	END_IF
END_CASE

//NCI Path ini Listeden Seçme Adımları
//NC kodunun oldugu klasördeki .nc leri listeleme
fbFindFileList(
	sNetId			:= '', 
	sPathName		:= sPathName, 
	eCmd			:= eEnumCmd_First, 
	pFindList		:= ADR(arrFileList), 
	cbFindList		:= SIZEOF(arrFileList), 
	bExecute		:= bExecuteFindList, 
	tTimeout		:= T#3S);

//3 sn de bir Liste Güncelleme 
tUpdatePathList(IN:= (NOT tUpdatePathList.Q) AND (NOT bChangeFile) , PT:= T#3S);
IF tUpdatePathList.Q THEN 
	bExecuteFindList	:= TRUE;
ELSE
	bExecuteFindList	:= FALSE;
END_IF
	
//Liste Seçiminde Select ve Cancel a Göre Seçili Öğeyi Ayarlama
//Eğer Ayarlanmasaydı Listeye Tekrar Girildiğinde Cancel Edilince Seçili Değil En Son Tıklanan Aktif Kalıyordu
CASE nStateFileNameList OF 
0:
	IF bChangeFile THEN 
		nLastFileNameList	:= nFileNameList;
		nStateFileNameList	:= 10;
	END_IF

10:
	IF bSelectFile THEN 
		nLastFileNameList	:= nFileNameList;
		nStateFileNameList	:= 20;
	ELSIF bCancelSelectFile THEN 
		nFileNameList		:= nLastFileNameList;
		nStateFileNameList	:= 20;
	END_IF

20:
	IF NOT bSelectFile THEN 
		nStateFileNameList	:= 0;
	END_IF
END_CASE

//ST_FindFileEntry tipinin içerisinden sadece ismi çekme 
FOR i:=0 TO 19 BY 1 DO 
	arrFileNameList[i]	:= arrFileList[i].sFileName;
END_FOR

//Path Seçim Ekranındaki Pathi Aktif Etme 
IF bSelectFile THEN 
	sFileName	:= CONCAT('C:\TwinCAT\CNC\',arrFileNameList[nFileNameList+1]);
	//Path in HMI Ekranında görüntülenecek hali
	sFileNameVisu	:= arrFileNameList[nFileNameList+1];
END_IF
END_ACTION

END_PROGRAM

// ---- POUs/UTIL/FB_Flash.TcPOU
FUNCTION_BLOCK FB_Flash
VAR_INPUT
	bEnable		: BOOL;
	tInterval	: TIME;
END_VAR
VAR_OUTPUT
	Q			: BOOL;
END_VAR
VAR
	tWait		: TON;
END_VAR


tWait(IN:= bEnable AND NOT tWait.Q  , PT:= tInterval);

IF bEnable THEN
	IF tWait.ET > (tInterval / 2) THEN
		Q	:= TRUE;
	ELSE
		Q	:= FALSE;
	END_IF
ELSE
	Q	:= FALSE;
END_IF

END_FUNCTION_BLOCK

// ---- VISUs/AxisList/VisuAxisX.TcVIS
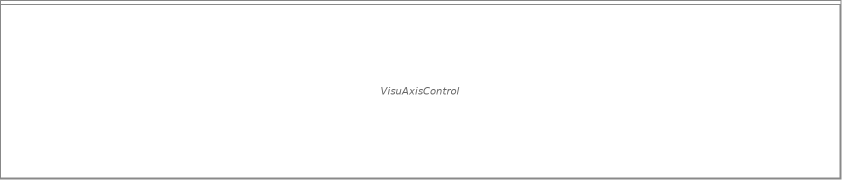
VISUALIZATION VisuAxisX  // 842x180
    Frame (0,4 840x174)
        shows VisuAxisControl(sAxisName := sAxisXName, stAxisVisu := stAxisX)
END_VISUALIZATION

// ---- VISUs/AxisList/VisuAxisZ.TcVIS
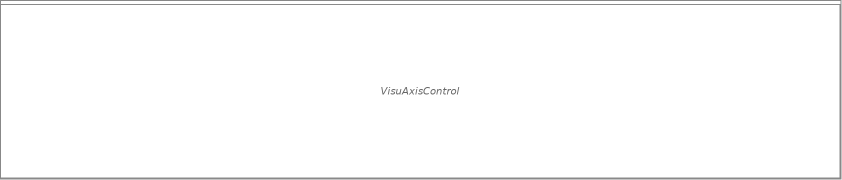
VISUALIZATION VisuAxisZ  // 842x180
    Frame (0,4 840x174)
        shows VisuAxisControl(sAxisName := sAxisZName, stAxisVisu := stAxisZ)
END_VISUALIZATION

// ---- VISUs/AxisList/VisuAxisZ_1.TcVIS
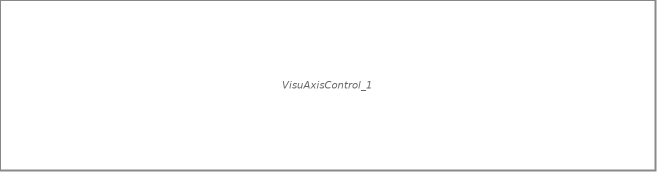
VISUALIZATION VisuAxisZ_1  // 657x172
    Frame (0,0 655x170)
        shows VisuAxisControl_1(sAxisName_1 := sAxisZName, stAxisVisu_1 := stAxisZ)
END_VISUALIZATION

// ---- VISUs/Frame/VisuAxisInfo.TcVIS
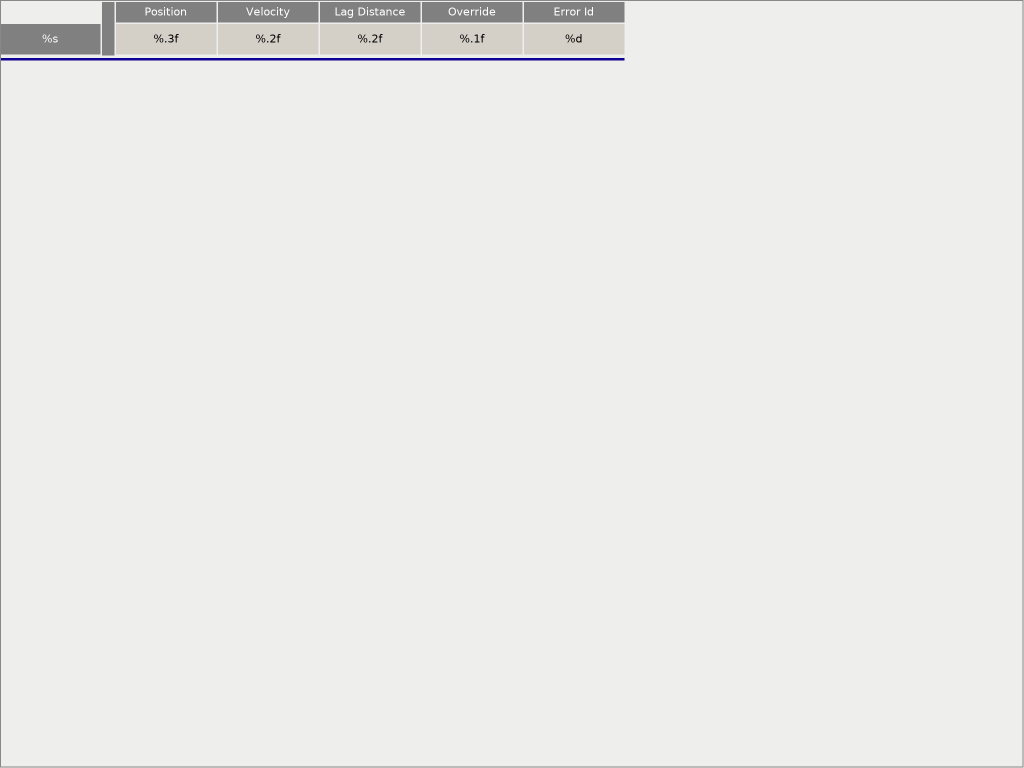
VISUALIZATION VisuAxisInfo  // 1024x768
VAR_IN_OUT
	sAxisName		: STRING;
	stAxisRefVisu	: AXIS_REF;
END_VAR
    Rectangle (0,24 100x30), "%s", text variable: sAxisName
    Rectangle (116,24 100x30), "%.3f", text variable: stAxisRefVisu.NcToPlc.ActPos
    Rectangle (116,2 100x20), "Position"
    Rectangle (218,24 100x30), "%.2f", text variable: stAxisRefVisu.NcToPlc.ActVelo
    Rectangle (422,24 100x30), "%.1f", text variable: stAxisRefVisu.PlcToNc.Override / 10000
    Rectangle (218,2 100x20), "Velocity"
    Rectangle (422,2 100x20), "Override"
    Rectangle (524,24 100x30), "%d", text variable: stAxisRefVisu.Status.ErrorID
    Rectangle (524,2 100x20), "Error Id"
    Rectangle (320,24 100x30), "%.2f", text variable: stAxisRefVisu.NcToPlc.PosDiff
    Rectangle (320,2 100x20), "Lag Distance"
    RoundedRectangle (102,2 12x53), colour toggle: stAxisRefVisu.Status.ControlLoopClosed
    RoundedRectangle (0,58 624x2)
END_VISUALIZATION

// ---- VISUs/GlobalTextList.TcGTLO
TEXTLIST GlobalTextList
  116 = ''
  114 = '           %s'
  113 = '      %s'
  115 = '  %s'
  37 = ' %s'
  74 = ' M1'
  76 = ' M3'
  77 = ' X'
  78 = ' Y'
  79 = ' Z'
  11 = '%.1f'
  8 = '%.2f'
  1 = '%.3f'
  96 = '%.3f mm/s'
  68 = '%a'
  13 = '%d'
  19 = '%s'
  69 = '%t %a'
  28 = '-->'
  27 = '<--'
  20 = 'Acceleration'
  117 = 'ACS'
  4 = 'Act. Position'
  9 = 'Act. Velocity'
  100 = 'AUTOMATIC MODE'
  18 = 'Axis'
  72 = 'Axis Coordinate System'
  32 = 'Axis Error'
  6 = 'Axis List'
  94 = 'Axis Reset'
  7 = 'Axis X'
  0 = 'Axis X '
  2 = 'Axis Y'
  3 = 'Axis Z'
  70 = 'Beckhoff Automation Turkey '
  26 = 'BW'
  112 = 'Cancel'
  55 = 'Cartesian Mode'
  110 = 'Checkbox'
  104 = 'Click for \nAuto Mode'
  105 = 'Click for \nManual Mode'
  21 = 'Deceleration'
  58 = 'DELTA ROBOT DEMOSET'
  93 = 'Drive Error'
  35 = 'Drive Reset'
  33 = 'DriveError'
  25 = 'Enable'
  12 = 'Error Id'
  43 = 'Finished'
  16 = 'Following Error'
  109 = 'G-Code List'
  29 = 'Home'
  24 = 'Home Pos'
  30 = 'Home Sensor'
  22 = 'Jerk'
  23 = 'Jog Velo'
  54 = 'Kin Execute'
  85 = 'KIN Group'
  56 = 'Kin Reset'
  53 = 'Kinematic Control'
  17 = 'Lag Distance'
  108 = 'Lag Distance[mm]'
  119 = 'Lag[mm]'
  80 = "M'"
  52 = 'M1_B'
  75 = 'M2'
  51 = 'M2_C'
  81 = 'M3'
  49 = 'M3_a'
  50 = 'M3_A'
  73 = 'Machine Coordinate System'
  71 = 'MAIN HMI '
  97 = 'Manual '
  101 = 'MANUAL MODE'
  92 = 'Manual Velocity'
  118 = 'MCS'
  95 = 'mm/s'
  87 = 'MODE'
  91 = 'MODE AUTOMATIC'
  89 = 'MODE MANUAL'
  90 = 'MODE OTOMATİK'
  31 = 'Move'
  38 = 'NCI Control'
  39 = 'NCI Enable'
  86 = 'NCI Group'
  45 = 'NCI Single'
  46 = 'NCI Single Mode'
  40 = 'NCI Start'
  47 = 'Next'
  36 = 'Open'
  57 = 'OpenFileDialog'
  88 = 'Otomatik'
  10 = 'Override'
  99 = 'Path'
  14 = 'Position'
  59 = 'POSITION M1'
  60 = 'Position M1'
  61 = 'Position M2'
  62 = 'Position M3'
  63 = 'Position X'
  64 = 'Position Y'
  65 = 'Position Z'
  106 = 'Position[mm]'
  67 = 'Power'
  102 = 'Press'
  103 = 'Press for \nAuto Mode'
  66 = 'R'
  34 = 'Reset'
  41 = 'Running'
  111 = 'Select'
  5 = 'Set. Position'
  48 = 'Single Mode'
  42 = 'Stopped'
  44 = 'Valve'
  15 = 'Velocity'
  107 = 'Velocity[mm/s]'
  98 = 'www.beckhoff.com.tr'
  82 = 'X'
  83 = 'Y'
  84 = 'Z'
END_TEXTLIST

// ---- VISUs/Visualization.TcVIS
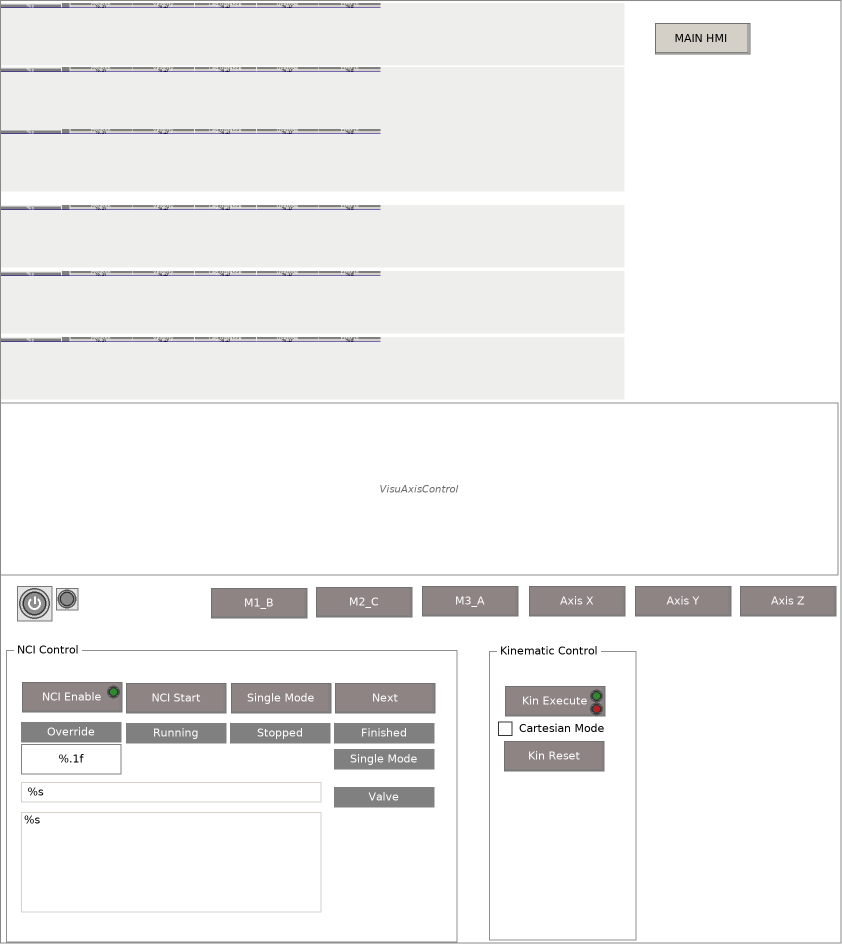
VISUALIZATION Visualization  // 842x944
    Frame (0,205 624x62)
        shows VisuAxisInfo(sAxisName := sAxisXName, stAxisRefVisu := AxisX)
    Frame (0,271 624x62)
        shows VisuAxisInfo(sAxisName := sAxisYName, stAxisRefVisu := AxisY)
    Frame (0,337 624x62)
        shows VisuAxisInfo(sAxisName := sAxisZName, stAxisRefVisu := AxisZ)
    Frame (0,399 840x178)
        shows VisuAxisX()
        shows VisuAxisY()
        shows VisuAxisZ()
        shows VisuAxisM1()
        shows VisuAxisM2()
        shows VisuAxisM3()
    Button (529,586 96x30), "Axis X"
        OnMouseClick: FrameSelectionChange Selection=SelectedFrame=c36eaae5-f889-4027-b551-56d3c927f334, GlobSel=AssignType=Directly, SelType=Locally
    Button (635,586 96x30), "Axis Y"
        OnMouseClick: FrameSelectionChange Selection=SelectedFrame=c36eaae5-f889-4027-b551-56d3c927f334, Selection=1, GlobSel=AssignType=Directly, SelType=Locally
    Button (740,586 96x30), "Axis Z"
        OnMouseClick: FrameSelectionChange Selection=SelectedFrame=c36eaae5-f889-4027-b551-56d3c927f334, Selection=2, GlobSel=AssignType=Directly, SelType=Locally
    GroupBox (6,642 451x300), "NCI Control"
        Button (16,40 100x30), "NCI Enable"
            toggle PRG_NcControl.bNciEnable
        Textfield (15,170 300x100), "%s", text variable: PRG_NcControl.sNciLines
        Button (225,41 100x30), "Single Mode"
            toggle PRG_NcControl.bNciSingleMode
        Rectangle (15,102 100x30), "%.1f", text variable: PRG_NcControl.fNciOverride
            OnMouseClick: write the text variable via VisuDialogs.Numpad
        Rectangle (15,80 100x20), "Override"
        Rectangle (120,81 100x20), "Running", colour toggle: PRG_NcControl.bProgramRunning
        Rectangle (224,81 100x20), "Stopped", colour toggle: PRG_NcControl.bProgramStopped
        Rectangle (328,81 100x20), "Finished", colour toggle: PRG_NcControl.bProgramFinished
        Rectangle (328,145 100x20), "Valve", colour toggle: PRG_MFuncControl.bTestValveOutput
        Button (120,41 100x30), "NCI Start"
            toggle PRG_NcControl.bNciStart
        Button (329,41 100x30), "Next"
            tap PRG_NcControl.bNciNextStep
        Rectangle (328,107 100x20), "Single Mode", colour toggle: PRG_NcControl.bSingleModeActive
        Lamp1 (100,42 15x16), variable: PRG_NcControl.bBuildGroupDone, style: Lamp-Lamp1-Green
    Textfield (21,782 300x20), "%s", text variable: PRG_NcControl.sNciActualLine
    Frame (0,3 624x62)
        shows VisuAxisInfo(sAxisName := sAxisM1_BName, stAxisRefVisu := AxisM1_B)
    Frame (0,67 624x62)
        shows VisuAxisInfo(sAxisName := sAxisM2_CName, stAxisRefVisu := AxisM2_C)
    Frame (0,129 624x62)
        shows VisuAxisInfo(sAxisName := sAxisM3_AName, stAxisRefVisu := AxisM3_A)
    Button (422,586 96x30), "M3_A"
        OnMouseClick: FrameSelectionChange Selection=SelectedFrame=c36eaae5-f889-4027-b551-56d3c927f334, Selection=5, GlobSel=AssignType=Directly, SelType=Locally
    Button (316,587 96x30), "M2_C"
        OnMouseClick: FrameSelectionChange Selection=SelectedFrame=c36eaae5-f889-4027-b551-56d3c927f334, Selection=4, GlobSel=AssignType=Directly, SelType=Locally
    Button (211,588 96x30), "M1_B"
        OnMouseClick: FrameSelectionChange Selection=SelectedFrame=c36eaae5-f889-4027-b551-56d3c927f334, Selection=3, GlobSel=AssignType=Directly, SelType=Locally
    GroupBox (489,643 147x297), "Kinematic Control"
        Button (16,43 100x30), "Kin Execute"
            tap PRG_Kinematic.bExecuteKinConfigGroup
        Checkbox (7,76 119x19), "Cartesian Mode", variable: PRG_Kinematic.bCartesianMode
        Button (15,98 100x30), "Kin Reset"
            tap PRG_Kinematic.bExecuteKinResetGroup
        Lamp1 (100,45 15x16), variable: PRG_Kinematic.fbKinConfigGroup.eKinStatus = KinStatus_Ready, style: Lamp-Lamp1-Green
        Lamp1 (100,58 15x16), variable: PRG_Kinematic.fbKinConfigGroup.bError, invisible if: not PRG_Kinematic.fbKinConfigGroup.bError, style: Lamp-Lamp1-Red
    PowerSwitch (17,586 35x35), variable: GVL_Process.bAllAxesEnable, behaviour: TOGGLE, style: Switch-PowerSwitch-Gray
    PushSwitch (54,588 26x22), variable: GVL_Process.bAllAxesReset, behaviour: TAP, style: Switch-PushSwitch-Gray
    Button (655,23 95x31), "MAIN HMI"
        OnMouseClick: change screen: Visualization_AxesInfo_Manual
END_VISUALIZATION
